// TIA Portal V19 program export: 0 tag tables, 0 data types, 5 data blocks, 88 code blocks (in call order from the OBs), 6 instance data blocks

DATA_BLOCK "DB_System"   // DB3
{ S7_Optimized_Access := 'TRUE' }
// stored: AutoNumber false, MemoryReserve 100
   VAR
      datetime : Struct
         current : DTL := DTL#2025-09-17-14:58:30.265837800;
      END_STRUCT;
      firstCycle : Bool := TRUE;
      reqPointers : Bool := FALSE;
      reqParametrizations : Bool := FALSE;
   END_VAR
   VAR RETAIN
      modulesGroup : Struct
         ADIN { S7_SetPoint := 'True'} : Bool := FALSE;
         AIN { S7_SetPoint := 'True'} : Bool := TRUE;
         DIFF { S7_SetPoint := 'True'} : Bool := FALSE;
         DIN { S7_SetPoint := 'True'} : Bool := TRUE;
         MTR { S7_SetPoint := 'True'} : Bool := TRUE;
         MTRDIR { S7_SetPoint := 'True'} : Bool := TRUE;
         MTRLIN { S7_SetPoint := 'True'} : Bool := FALSE;
         VLV { S7_SetPoint := 'True'} : Bool := FALSE;
         CVLV { S7_SetPoint := 'True'} : Bool := FALSE;
      END_STRUCT;
   END_VAR
   VAR
      reqQuickSetup { S7_SetPoint := 'True'} : "modTypes";
   END_VAR
BEGIN
   reqQuickSetup.adin := FALSE;
   reqQuickSetup.ain := FALSE;
   reqQuickSetup.cvlv := FALSE;
   reqQuickSetup.din := FALSE;
   reqQuickSetup.mtr := FALSE;
   reqQuickSetup.mtrDir := FALSE;
   reqQuickSetup.mtrLin := FALSE;
   reqQuickSetup.vlv := FALSE;
END_DATA_BLOCK

DATA_BLOCK "FAULTS"   // DB14
{ S7_Optimized_Access := 'FALSE' }
   VAR
      ADIN { S7_SetPoint := 'True'} : Array[0.."MAX_ADIN"] of "UDT_DINFAULTS";   // ADIN = 1 alarm/instance, 24 x 8 (each type contains 8 instances) = 192 alarms, offset = 0
      AIN { S7_SetPoint := 'True'} : Array[0.."MAX_AIN"] of "UDT_AINFAULTS";   // AIN = 2 alarms/instance, 200 x 2 = 400 alarms, offset = 192
      DIFF { S7_SetPoint := 'True'} : Array[0.."MAX_DIFF"] of "UDT_AINFAULTS";   // DIFF = 2 alarms/instance, 32 x 2 = 64 alarms, offset = 592
      DIN { S7_SetPoint := 'True'} : Array[0.."MAX_DIN"] of "UDT_DINFAULTS";   // DIN = 1 alarm/instance, 24 x 8 (each type contains 8 instances) = 192 alarms, offset = 656
      MTR { S7_SetPoint := 'True'} : Array[0.."MAX_MTR"] of "UDT_MTRFAULTS";   // MTR = 6 alarms/instance, 200 x 6 = 1200 alarms, offset = 848
      MTRLIN { S7_SetPoint := 'True'} : Array[0.."MAX_MTRLIN"] of "UDT_MTRFAULTS";   // MTRLIN = 6 alarms/instance, 80 x 6 = 480 alarms, offset = 2048
      MTRDIR { S7_SetPoint := 'True'} : Array[0.."MAX_MTRDIR"] of "UDT_MTRFAULTS";   // MTRDIR = 6 alarms/instance, 200 x 6 = 1200 alarms, offset = 2528
      VLV { S7_SetPoint := 'True'} : Array[0.."MAX_VLV"] of "UDT_VALVEFAULTS";   // VLV = 4 alarms/instance, 200 x 6 = 1200 alarms, offset = 3728
      Plant { S7_SetPoint := 'True'} : Array[0.."MAX_PLANT"] of "UDT_DINFAULTS";   // Plant = 1 alarm/instance, 24 x 8 (each type contains 8 instances) = 192 alarms, offset = 4928
   END_VAR
BEGIN
END_DATA_BLOCK

DATA_BLOCK "MODULES_CTRL"   // DB54
{ S7_Optimized_Access := 'TRUE' }
// stored: MemoryReserve 100
   VAR
      ADIN { ExternalAccessible := 'False'; ExternalVisible := 'False'; ExternalWritable := 'False'; S7_SetPoint := 'True'} : Array[0.."M_ADIN"] of "CTRL_ADIN";
      AIN { ExternalAccessible := 'False'; ExternalVisible := 'False'; ExternalWritable := 'False'; S7_SetPoint := 'True'} : Array[0.."M_AIN"] of "CTRL_AIN";
      CVLV { ExternalAccessible := 'False'; ExternalVisible := 'False'; ExternalWritable := 'False'; S7_SetPoint := 'True'} : Array[0.."M_CVLV"] of "CTRL_CVLV";
      DIFF { ExternalAccessible := 'False'; ExternalVisible := 'False'; ExternalWritable := 'False'; S7_SetPoint := 'True'} : Array[0.."M_DIFF"] of "CTRL_DIFF";
      DIN { ExternalAccessible := 'False'; ExternalVisible := 'False'; ExternalWritable := 'False'; S7_SetPoint := 'True'} : Array[0.."M_DIN"] of "CTRL_DIN";
      MTRDIR { ExternalAccessible := 'False'; ExternalVisible := 'False'; ExternalWritable := 'False'; S7_SetPoint := 'True'} : Array[0.."M_MTRDIR"] of "CTRL_MTRDIR";
      MTRLIN { ExternalAccessible := 'False'; ExternalVisible := 'False'; ExternalWritable := 'False'; S7_SetPoint := 'True'} : Array[0.."M_MTRLIN"] of "CTRL_MTRLIN";
      MTR { ExternalAccessible := 'False'; ExternalVisible := 'False'; ExternalWritable := 'False'; S7_SetPoint := 'True'} : Array[0.."M_MTR"] of "CTRL_MTR";
      VLV { ExternalAccessible := 'False'; ExternalVisible := 'False'; ExternalWritable := 'False'; S7_SetPoint := 'True'} : Array[0.."M_VLV"] of "CTRL_VLV";
   END_VAR
BEGIN
END_DATA_BLOCK

DATA_BLOCK "WARNINGS"   // DB15
{ S7_Optimized_Access := 'FALSE' }
   VAR
      AIN { S7_SetPoint := 'True'} : Array[0.."MAX_AIN"] of "UDT_AINWARNS";   // AIN = 2 alarms/instance, 200 x 2 = 400 alarms, offset = 8000
      DIFF { S7_SetPoint := 'True'} : Array[0.."MAX_DIFF"] of "UDT_AINWARNS";   // DIFF = 2 alarms/instance, 200 x 2 = 400 alarms, offset = 8400
      Plant { S7_SetPoint := 'True'} : Array[0.."MAX_PLANT"] of "UDT_DINFAULTS";   // Plant = 1 alarm/instance, 24 x 8 (each type contains 8 instances) = 192 alarms, offset = 8800
   END_VAR
BEGIN
END_DATA_BLOCK

DATA_BLOCK "SpProd"   // DB220
{ S7_Optimized_Access := 'TRUE' }
AUTHOR : CH
FAMILY : Aktina
NAME : SEQUENCE
// stored: AutoNumber false, MemoryReserve 100
   VAR RETAIN
      drill { S7_SetPoint := 'True'} : "dtDrill";
      supply : "dtSupply";
   END_VAR
   VAR
      iTank { S7_SetPoint := 'True'} : Array[0..1] of "UDT_TANKPRESS_2";
      autoReset { S7_SetPoint := 'True'} : Array[0..0] of "dtAutoReset";
   END_VAR
BEGIN
   drill.level[0] := 75;
   drill.level[1] := 85;
   drill.level[2] := 90;
   drill.level[3] := 100;
   drill.tDelay := T#5S;
   drill.setPriority[0] := 2;
   drill.setPriority[1] := 3;
   drill.setPriority[2] := 0;
   drill.loadPriority[0] := 2;
   drill.loadPriority[1] := 3;
   drill.loadPriority[2] := 0;
   drill.TankAvailable[0..1] := TRUE;
   drill.loadBtn := FALSE;
   supply.setAvailPumps[0] := FALSE;
   supply.setAvailPumps[1..3] := TRUE;
   supply.loadAvailPumps[0] := FALSE;
   supply.loadAvailPumps[1..3] := TRUE;
   supply.availPumps[0..2] := TRUE;
   supply.loadBtn := FALSE;
   supply.pressureSP := 4.0;
   supply.hhPressureAlm := 6.0;
   supply.highFlow := 35.0;
   supply.lowFlow := 10.0;
   supply.zChangeThr := 0.3;
   supply.zChangeDelay := T#1S;
   supply.PumpInterval := T#10H;
   supply.zoneChangeOP := 90.0;
   supply.overlapDelay := T#10S;
   supply.downgradeDelay := T#40S;
   supply.chLead := 2;
   supply.enRotation := FALSE;
   supply.stageUp.zoneChangeOP := 95.0;
   supply.stageUp.delayUpgrade := T#5S;
   // supply.stageDown[0] : bigPump
   // supply.stageDown[1] : midPump
   // supply.stageDown[2] : smallPump
   supply.stageDown[0..3].zoneChangeOP := 40.0;
   supply.stageDown[0..3].prevOP := 20.0;
   supply.stageDown[0..3].nextOP := 70.0;
   supply.stageDown[0].stabilizeDelay := T#1M;
   supply.stageDown[1].stabilizeDelay := T#10S;
   supply.stageDown[2..3].stabilizeDelay := T#5S;
   supply.stageDown[0..3].followUp := FALSE;
   iTank[0..1].r := 1.0;
   iTank[0..1].d := 263.0;
   iTank[0..1].hPt := 0.0;
   iTank[0..1].hBase := 0.0;
   iTank[0..1].hCyl := 525.0;
   iTank[0].hAct := 465.6394;
   iTank[1].hAct := 463.0353;
   iTank[0].vol := 25295.94;
   iTank[1].vol := 25154.47;
   // autoReset[0] : Grid
   autoReset[0].maxAlarms := 10;
   autoReset[0].perT := T#1H;
   autoReset[0].autoresetT := T#30S;
END_DATA_BLOCK

ORGANIZATION_BLOCK "Main"   // OB1, LAD, ProgramCycle
TITLE = "Main Program Sweep (Cycle)"
{ S7_Optimized_Access := 'TRUE' }
// stored: SetENOAutomatically false
   VAR_INPUT
      Initial_Call : Bool;   // Initial call of this OB
      Remanence : Bool;   // =True, if remanent data are available
   END_VAR
BEGIN
END_ORGANIZATION_BLOCK

ORGANIZATION_BLOCK "Cyclic interrupt 100ms"   // OB30, LAD, CyclicInterrupt
{ S7_Optimized_Access := 'TRUE' }
// stored: SetENOAutomatically false
   VAR_INPUT
      Initial_Call : Bool;   // Initial call of this OB
      Event_Count : Int;   // Events discarded
   END_VAR
   VAR_TEMP
      i : Int;
   END_VAR
BEGIN
END_ORGANIZATION_BLOCK

ORGANIZATION_BLOCK "Diagnostic error interrupt"   // OB82, LAD, DiagnosticErrorInterrupt
{ S7_Optimized_Access := 'TRUE' }
// stored: SetENOAutomatically false
   VAR_INPUT
      IO_State : Word;   // IO state of the HW object
      LADDR : HW_ANY;   // Hardware identifier
      Channel : UInt;   // Channel number
      MultiError : Bool;   // =true if more than one error is present
   END_VAR
BEGIN
END_ORGANIZATION_BLOCK

ORGANIZATION_BLOCK "Pull or plug of modules"   // OB83, LAD, PullOrPlugOfModules
{ S7_Optimized_Access := 'TRUE' }
// stored: SetENOAutomatically false
   VAR_INPUT
      LADDR : HW_IO;   // Hardware identifier
      Event_Class : Byte;   // 16#38/39: module inserted, removed
      Fault_ID : Byte;   // Fault identifier
   END_VAR
BEGIN
END_ORGANIZATION_BLOCK

ORGANIZATION_BLOCK "Rack or station failure"   // OB86, LAD, RackOrStationFailure
{ S7_Optimized_Access := 'TRUE' }
// stored: SetENOAutomatically false
   VAR_INPUT
      LADDR : HW_DEVICE;   // Hardware identifier
      Event_Class : Byte;   // Event class
      Fault_ID : Byte;   // Fault identifier
   END_VAR
BEGIN
END_ORGANIZATION_BLOCK

ORGANIZATION_BLOCK "Time error interrupt"   // OB80, LAD, TimeErrorInterrupt
{ S7_Optimized_Access := 'TRUE' }
// stored: SetENOAutomatically false
   VAR_INPUT
      Fault_ID : Byte;   // Fault identifier
      Csg_OBnr : OB_ANY;   // Number of OB causing the error
      Csg_Prio : UInt;   // Priority of OB causing the error
   END_VAR
BEGIN
END_ORGANIZATION_BLOCK

FUNCTION_BLOCK "AFB_Totalizer"   // FB3, LAD
{ S7_Optimized_Access := 'TRUE' }
// stored: MemoryReserve 100, SetENOAutomatically false
   VAR_INPUT
      inputVolume { ExternalAccessible := 'False'; ExternalVisible := 'False'; ExternalWritable := 'False'} : Real;
      startBtn { ExternalAccessible := 'False'; ExternalVisible := 'False'; ExternalWritable := 'False'} : Bool;
      stopBtn { ExternalAccessible := 'False'; ExternalVisible := 'False'; ExternalWritable := 'False'} : Bool;
   END_VAR
   VAR_OUTPUT
      addedVolume { ExternalAccessible := 'False'; ExternalVisible := 'False'; ExternalWritable := 'False'} : Real;
      tempCount { ExternalAccessible := 'False'; ExternalVisible := 'False'; ExternalWritable := 'False'} : Bool;
   END_VAR
   VAR
      previousVolume { ExternalAccessible := 'False'; ExternalVisible := 'False'; ExternalWritable := 'False'} : Real;
      Start_Trigger { S7_SetPoint := 'True'} : R_TRIG;
      Strop_Trigger { S7_SetPoint := 'True'} : R_TRIG;
   END_VAR
BEGIN

REGION Network 1
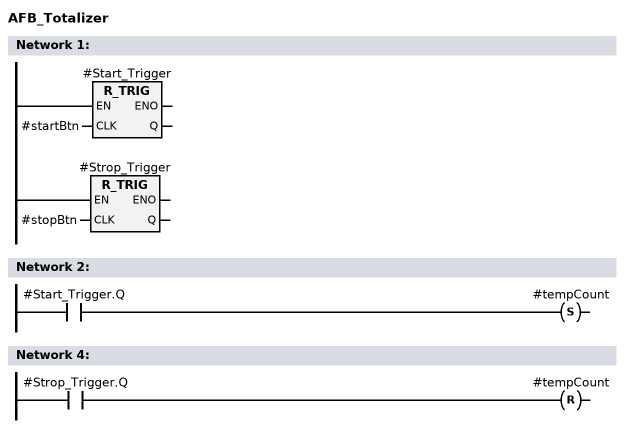
   RUNG wire#powerrail
      #Start_Trigger.R_TRIG(CLK := #startBtn, Q =>)
   END_RUNG
   RUNG wire#powerrail
      #Strop_Trigger.R_TRIG(CLK := #stopBtn, Q =>)
   END_RUNG
   // the same network as SCL:
   #Start_Trigger(CLK := #startBtn);   // R_TRIG
   #Strop_Trigger(CLK := #stopBtn);   // R_TRIG
END_REGION

REGION Network 2
   RUNG wire#powerrail
      Contact( #Start_Trigger.Q )
      S_Coil( #tempCount )
   END_RUNG
   // the same network as SCL:
   IF #Start_Trigger.Q THEN #tempCount := TRUE; END_IF;
END_REGION

REGION Network 3 (SCL)

   IF #startBtn THEN
       #previousVolume := #inputVolume;
   END_IF;


   IF #tempCount THEN

       #addedVolume := #inputVolume - #previousVolume;
       ;
   ELSE
       #addedVolume := 0 ;
   END_IF;
END_REGION

REGION Network 4
   RUNG wire#powerrail
      Contact( #Strop_Trigger.Q )
      R_Coil( #tempCount )
   END_RUNG
   // the same network as SCL:
   IF #Strop_Trigger.Q THEN #tempCount := FALSE; END_IF;
END_REGION
END_FUNCTION_BLOCK

FUNCTION "AFC_Counter" : Void   // FC1, FBD
TITLE = AFC_COUNTER
{ S7_Optimized_Access := 'TRUE' }
AUTHOR : CH
FAMILY : Aktina
NAME : Global
// AFC_COUNTER
// stored: AutoNumber false, IsIECCheckEnabled true, SetENOAutomatically false
   VAR_INPUT
      Trigger : Bool;
      Pulse : Bool;
      Reset : Bool;
   END_VAR
   VAR_IN_OUT
      Data : Variant;
   END_VAR
   VAR_TEMP
      i : "UDT_COUNTER";
      logical1 : Bool;
   END_VAR
BEGIN

REGION Network 1: GEN: Set Logical 1
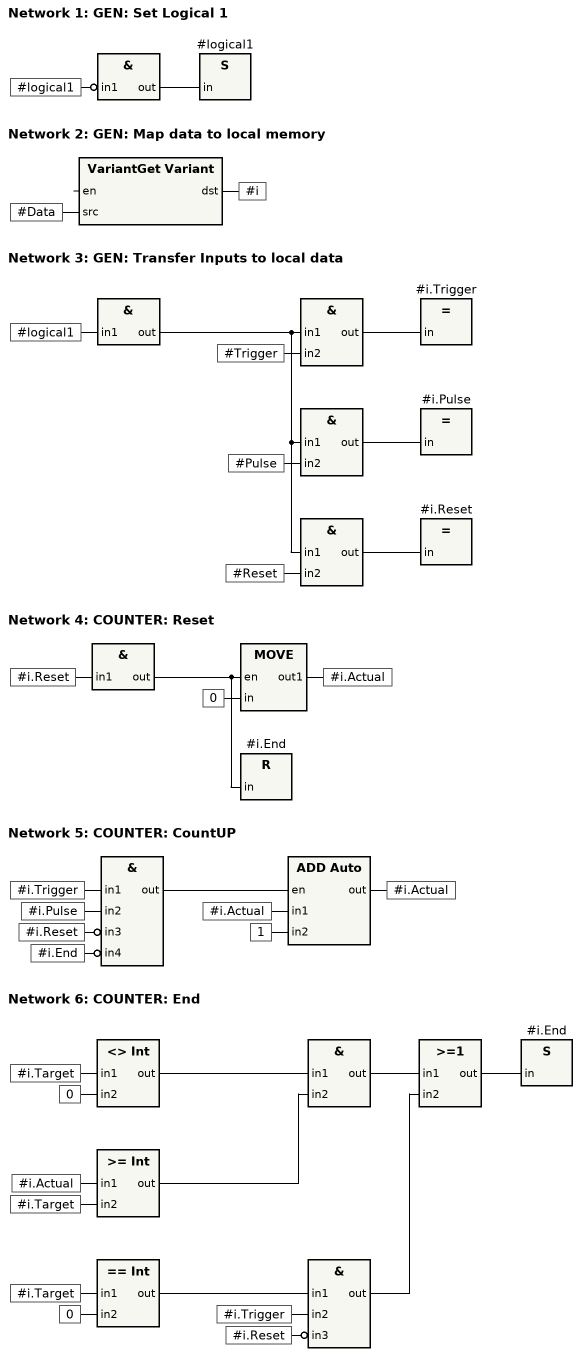
   IF NOT #logical1 THEN #logical1 := TRUE; END_IF;
END_REGION

REGION Network 2: GEN: Map data to local memory
   // no SCL statement known for VariantGet: written as a call
   VariantGet(src := #Data, dst => #i);
END_REGION

REGION Network 3: GEN: Transfer Inputs to local data
   #i.Trigger := #logical1 AND #Trigger;
   #i.Pulse := #logical1 AND #Pulse;
   #i.Reset := #logical1 AND #Reset;
END_REGION

REGION Network 4: COUNTER: Reset
   IF #i.Reset THEN
       #i.Actual := 0;
       #i.End := FALSE;
   END_IF;
END_REGION

REGION Network 5: COUNTER: CountUP
   IF #i.Trigger AND #i.Pulse AND NOT #i.Reset AND NOT #i.End THEN #i.Actual := #i.Actual + 1; END_IF;
END_REGION

REGION Network 6: COUNTER: End
   IF ((#i.Target <> 0) AND (#i.Actual >= #i.Target)) OR ((#i.Target = 0) AND #i.Trigger AND NOT #i.Reset) THEN
       #i.End := TRUE;
   END_IF;
END_REGION

REGION Network 7: COUNTER: Calculate Remaining
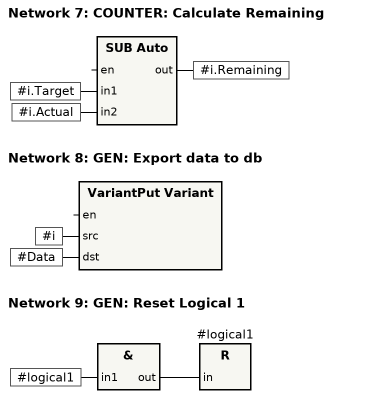
   #i.Remaining := #i.Target - #i.Actual;
END_REGION

REGION Network 8: GEN: Export data to db
   // no SCL statement known for VariantPut: written as a call
   VariantPut(src := #i, dst := #Data);
END_REGION

REGION Network 9: GEN: Reset Logical 1
   IF #logical1 THEN #logical1 := FALSE; END_IF;
END_REGION
END_FUNCTION

FUNCTION "AFC_DelayON" : Void   // FC2, FBD
TITLE = AFC_DELAYON
{ S7_Optimized_Access := 'TRUE' }
AUTHOR : CH
FAMILY : Aktina
NAME : Global
// AFC_DELAYON
// stored: AutoNumber false, IsIECCheckEnabled true, SetENOAutomatically false
   VAR_INPUT
      cmd : Bool;   // Command run
      Pulse : Bool;   // 100ms pulse
      Reset : Bool;   // Reset immediately
   END_VAR
   VAR_OUTPUT
      on : Bool;   // Activation
   END_VAR
   VAR_IN_OUT
      Data : Variant;   // Data area
   END_VAR
   VAR_TEMP
      i : "UDT_DELAYON";   // Local stack
      logical1 : Bool;   // Logical 1
      calc : Real;   // Calculation intermediate
   END_VAR
BEGIN

REGION Network 1: GEN: Set Logical 1
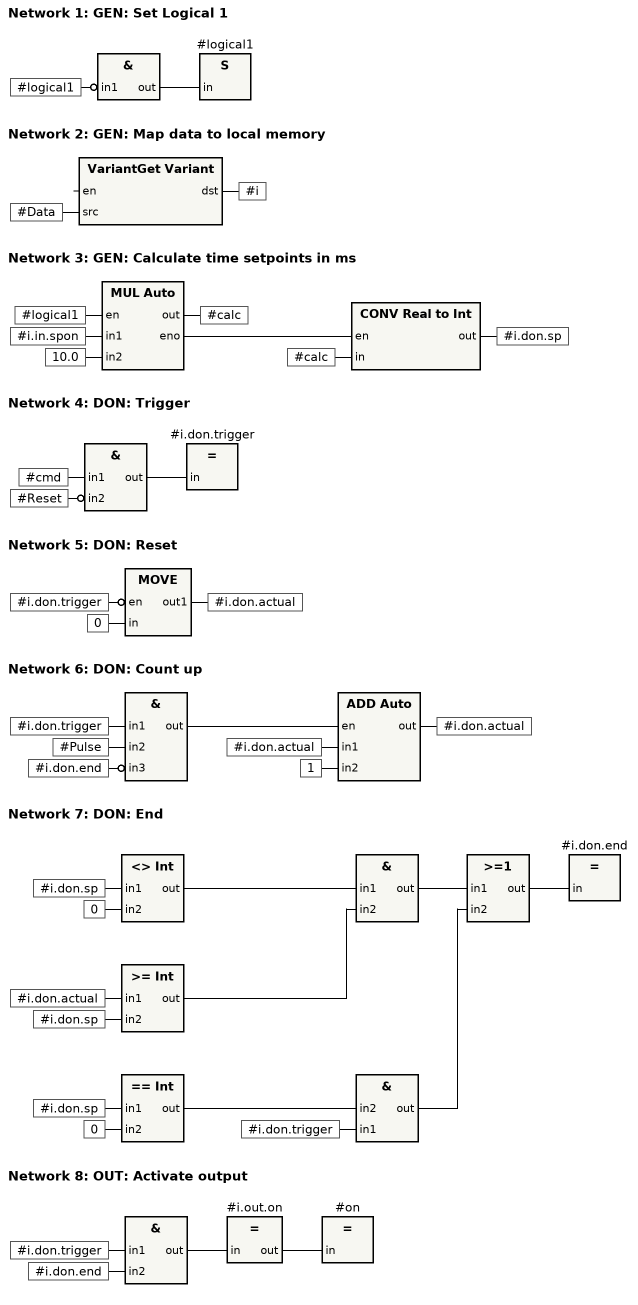
   IF NOT #logical1 THEN #logical1 := TRUE; END_IF;
END_REGION

REGION Network 2: GEN: Map data to local memory
   // no SCL statement known for VariantGet: written as a call
   VariantGet(src := #Data, dst => #i);
END_REGION

REGION Network 3: GEN: Calculate time setpoints in ms
   IF #logical1 THEN
       #calc := #i.in.spon * 10.0;
       #i.don.sp := REAL_TO_INT(#calc);
   END_IF;
END_REGION

REGION Network 4: DON: Trigger
   #i.don.trigger := #cmd AND NOT #Reset;
END_REGION

REGION Network 5: DON: Reset
   IF NOT #i.don.trigger THEN #i.don.actual := 0; END_IF;
END_REGION

REGION Network 6: DON: Count up
   IF #i.don.trigger AND #Pulse AND NOT #i.don.end THEN #i.don.actual := #i.don.actual + 1; END_IF;
END_REGION

REGION Network 7: DON: End
   #i.don.end := ((#i.don.sp <> 0) AND (#i.don.actual >= #i.don.sp)) OR ((#i.don.sp = 0) AND #i.don.trigger);
END_REGION

REGION Network 8: OUT: Activate output
   #i.out.on := #i.don.trigger AND #i.don.end;
   #on := #i.out.on;
END_REGION

REGION Network 9: GEN: Export data to db
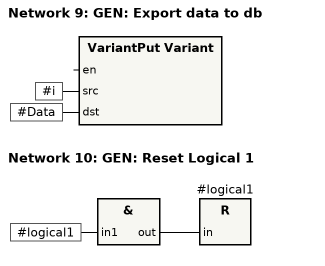
   // no SCL statement known for VariantPut: written as a call
   VariantPut(src := #i, dst := #Data);
END_REGION

REGION Network 10: GEN: Reset Logical 1
   IF #logical1 THEN #logical1 := FALSE; END_IF;
END_REGION
END_FUNCTION

FUNCTION "AFC_DelayONOFF" : Void   // FC4, FBD
TITLE = AFC_DELAYONOFF
{ S7_Optimized_Access := 'TRUE' }
AUTHOR : CH
FAMILY : Aktina
NAME : Global
// AFC_DELAYONOFF
// stored: AutoNumber false, IsIECCheckEnabled true, SetENOAutomatically false
   VAR_INPUT
      cmd : Bool;   // Command run
      Pulse : Bool;   // 100ms pulse
      Reset : Bool;   // Reset immediately
   END_VAR
   VAR_OUTPUT
      on : Bool;   // Activation
   END_VAR
   VAR_IN_OUT
      Data : Variant;   // Data area
   END_VAR
   VAR_TEMP
      i : "UDT_DELAYONOFF";   // Local stack
      logical1 : Bool;   // Logical 1
      calc : Real;   // Calculation intermediate
   END_VAR
BEGIN

REGION Network 1: GEN: Set Logical 1
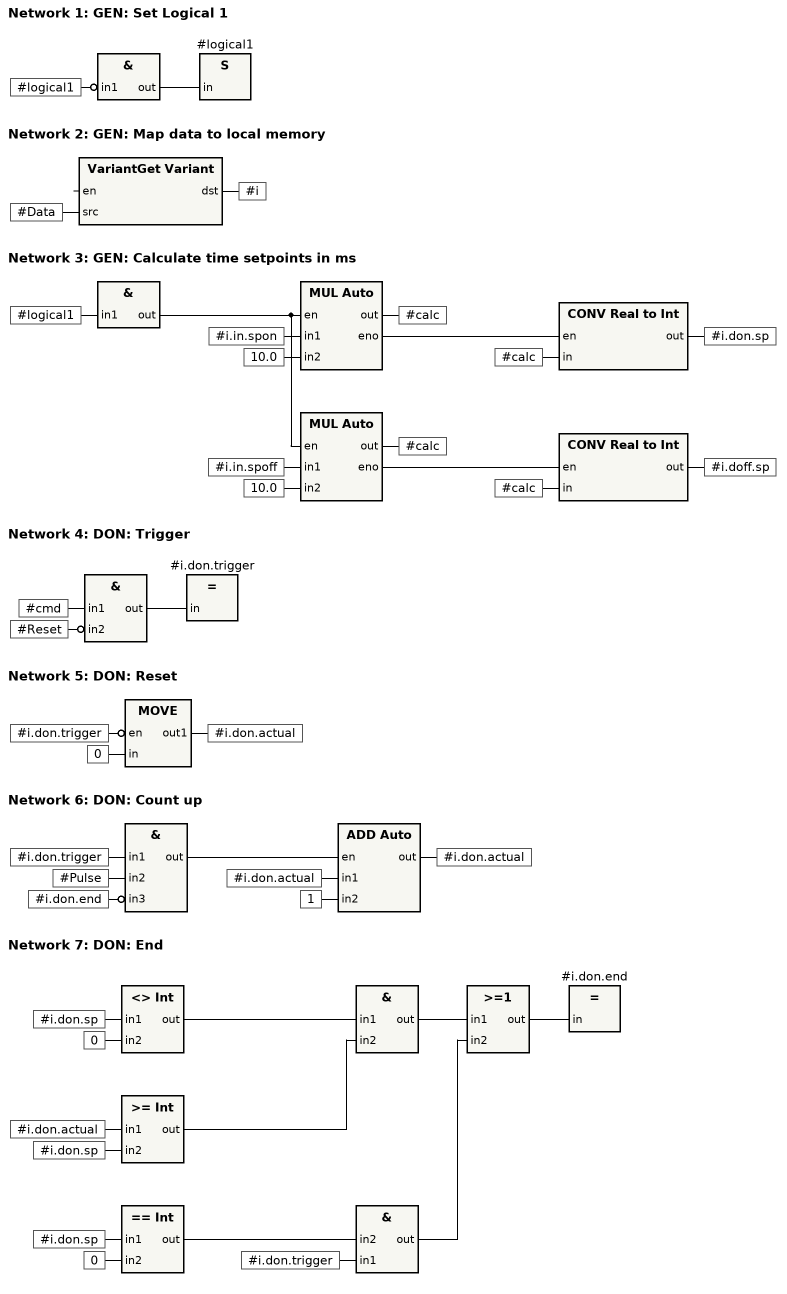
   IF NOT #logical1 THEN #logical1 := TRUE; END_IF;
END_REGION

REGION Network 2: GEN: Map data to local memory
   // no SCL statement known for VariantGet: written as a call
   VariantGet(src := #Data, dst => #i);
END_REGION

REGION Network 3: GEN: Calculate time setpoints in ms
   IF #logical1 THEN
       #calc := #i.in.spon * 10.0;
       #i.don.sp := REAL_TO_INT(#calc);
       #calc := #i.in.spoff * 10.0;
       #i.doff.sp := REAL_TO_INT(#calc);
   END_IF;
END_REGION

REGION Network 4: DON: Trigger
   #i.don.trigger := #cmd AND NOT #Reset;
END_REGION

REGION Network 5: DON: Reset
   IF NOT #i.don.trigger THEN #i.don.actual := 0; END_IF;
END_REGION

REGION Network 6: DON: Count up
   IF #i.don.trigger AND #Pulse AND NOT #i.don.end THEN #i.don.actual := #i.don.actual + 1; END_IF;
END_REGION

REGION Network 7: DON: End
   #i.don.end := ((#i.don.sp <> 0) AND (#i.don.actual >= #i.don.sp)) OR ((#i.don.sp = 0) AND #i.don.trigger);
END_REGION

REGION Network 8: DOFF: Trigger
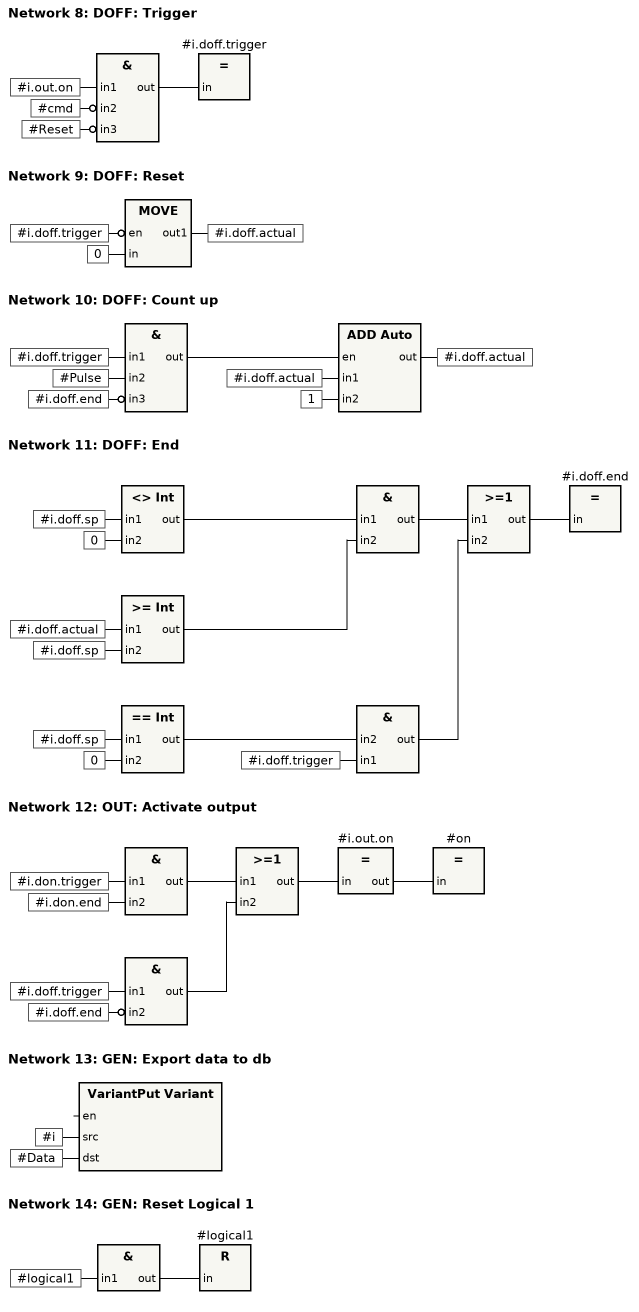
   #i.doff.trigger := #i.out.on AND NOT #cmd AND NOT #Reset;
END_REGION

REGION Network 9: DOFF: Reset
   IF NOT #i.doff.trigger THEN #i.doff.actual := 0; END_IF;
END_REGION

REGION Network 10: DOFF: Count up
   IF #i.doff.trigger AND #Pulse AND NOT #i.doff.end THEN #i.doff.actual := #i.doff.actual + 1; END_IF;
END_REGION

REGION Network 11: DOFF: End
   #i.doff.end := ((#i.doff.sp <> 0) AND (#i.doff.actual >= #i.doff.sp)) OR ((#i.doff.sp = 0) AND #i.doff.trigger);
END_REGION

REGION Network 12: OUT: Activate output
   #i.out.on := (#i.don.trigger AND #i.don.end) OR (#i.doff.trigger AND NOT #i.doff.end);
   #on := #i.out.on;
END_REGION

REGION Network 13: GEN: Export data to db
   // no SCL statement known for VariantPut: written as a call
   VariantPut(src := #i, dst := #Data);
END_REGION

REGION Network 14: GEN: Reset Logical 1
   IF #logical1 THEN #logical1 := FALSE; END_IF;
END_REGION
END_FUNCTION

FUNCTION "AFC_Steptimer" : Void   // FC35, FBD
TITLE = AFC_Steptimer
{ S7_Optimized_Access := 'TRUE' }
AUTHOR : CH
FAMILY : Aktina
NAME : Global
// AFC_Steptimer
// stored: AutoNumber false, SetENOAutomatically false
   VAR_INPUT
      "step" : Bool;   // Step activated
      count_max : Bool;   // Trigger for max step timer
      count_step : Bool;   // Trigger for conditional step timer
      Pulse : Bool;   // Pulse used for time count
      reset_max : Bool;   // Reset max step timer
      reset_step : Bool;   // Reset conditional step timer
      reset_warn : Bool;   // Reset max timer warning
   END_VAR
   VAR_OUTPUT
      max_warn : Bool;   // Max step timer has elapsed
   END_VAR
   VAR_IN_OUT
      Data : Variant;   // Unique data area for this counter
   END_VAR
   VAR_TEMP
      i : "UDT_STEPTIMER";
      logical1 : Bool;
      remain : UDInt;
      intermediate : UDInt;
      sec : UDInt;
      min : UDInt;
      hour : UDInt;
   END_VAR
BEGIN

REGION Network 1: GEN: Create Logical 1
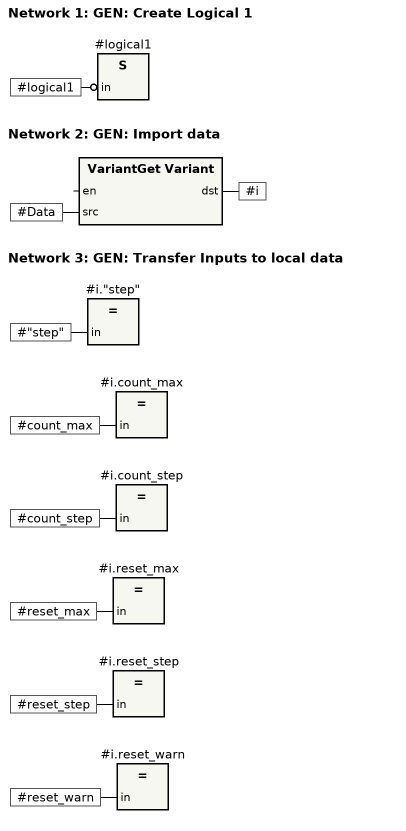
   IF NOT #logical1 THEN #logical1 := TRUE; END_IF;
END_REGION

REGION Network 2: GEN: Import data
   // no SCL statement known for VariantGet: written as a call
   VariantGet(src := #Data, dst => #i);
END_REGION

REGION Network 3: GEN: Transfer Inputs to local data
   #i."step" := #"step";
   #i.count_max := #count_max;
   #i.count_step := #count_step;
   #i.reset_max := #reset_max;
   #i.reset_step := #reset_step;
   #i.reset_warn := #reset_warn;
END_REGION

REGION Network 4: TIMER: Calculate seconds based on h, m, s (max)
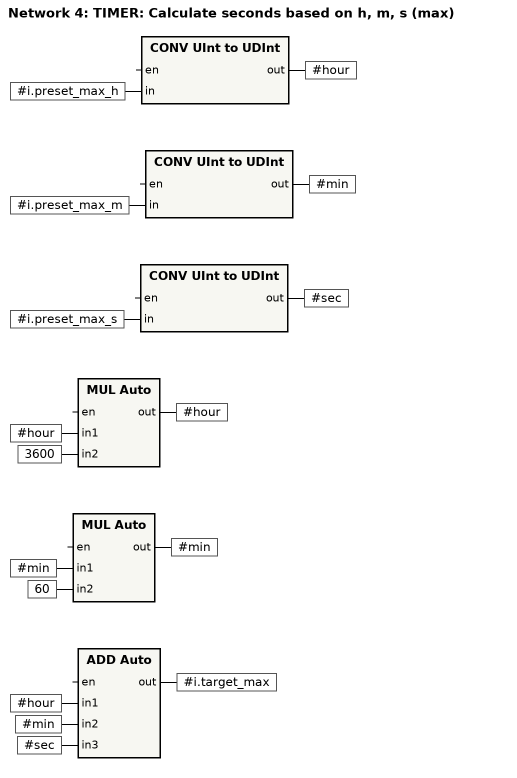
   #hour := UINT_TO_UDINT(#i.preset_max_h);
   #min := UINT_TO_UDINT(#i.preset_max_m);
   #sec := UINT_TO_UDINT(#i.preset_max_s);
   #hour := #hour * 3600;
   #min := #min * 60;
   #i.target_max := #hour + #min + #sec;
END_REGION

REGION Network 5: TIMER: Calculate seconds based on h, m, s (step)
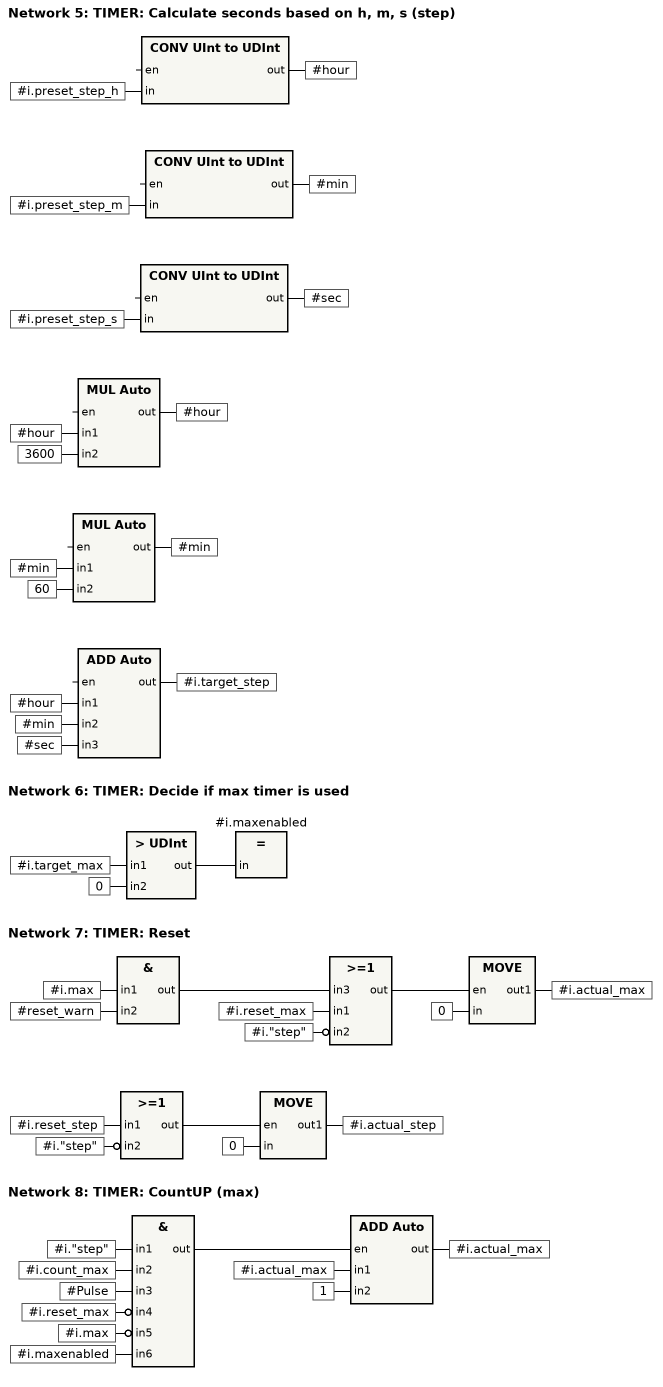
   #hour := UINT_TO_UDINT(#i.preset_step_h);
   #min := UINT_TO_UDINT(#i.preset_step_m);
   #sec := UINT_TO_UDINT(#i.preset_step_s);
   #hour := #hour * 3600;
   #min := #min * 60;
   #i.target_step := #hour + #min + #sec;
END_REGION

REGION Network 6: TIMER: Decide if max timer is used
   #i.maxenabled := #i.target_max > 0;
END_REGION

REGION Network 7: TIMER: Reset
   IF (#i.max AND #reset_warn) OR #i.reset_max OR NOT #i."step" THEN #i.actual_max := 0; END_IF;
   IF #i.reset_step OR NOT #i."step" THEN #i.actual_step := 0; END_IF;
END_REGION

REGION Network 8: TIMER: CountUP (max)
   IF #i."step" AND #i.count_max AND #Pulse AND NOT #i.reset_max AND NOT #i.max AND #i.maxenabled THEN
       #i.actual_max := #i.actual_max + 1;
   END_IF;
END_REGION

REGION Network 9: TIMER: CountUP (step)
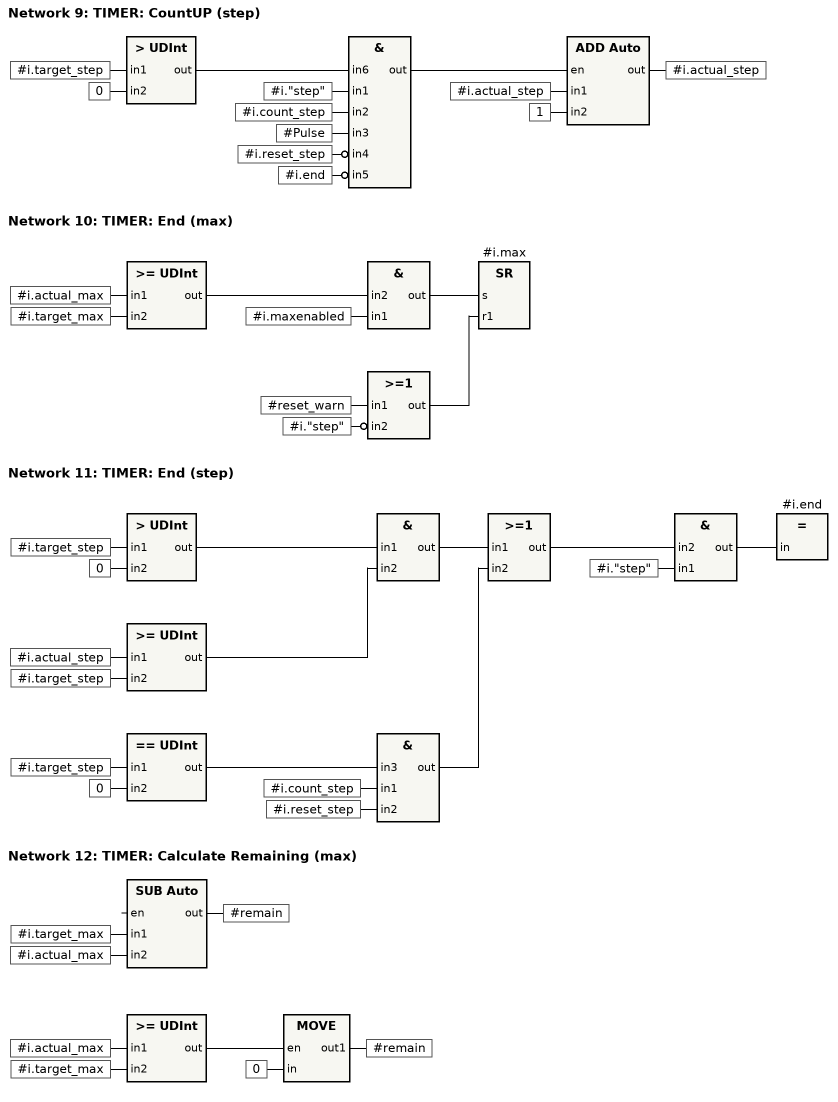
   IF (#i.target_step > 0) AND #i."step" AND #i.count_step AND #Pulse AND NOT #i.reset_step AND NOT #i.end THEN
       #i.actual_step := #i.actual_step + 1;
   END_IF;
END_REGION

REGION Network 10: TIMER: End (max)
   IF (#i.actual_max >= #i.target_max) AND #i.maxenabled THEN
       #i.max := TRUE;   // SR flip-flop
   END_IF;
   IF #reset_warn OR NOT #i."step" THEN #i.max := FALSE; END_IF;
END_REGION

REGION Network 11: TIMER: End (step)
   #i.end := (((#i.target_step > 0) AND (#i.actual_step >= #i.target_step)) OR ((#i.target_step = 0) AND #i.count_step AND #i.reset_step)) AND #i."step";
END_REGION

REGION Network 12: TIMER: Calculate Remaining (max)
   #remain := #i.target_max - #i.actual_max;
   IF #i.actual_max >= #i.target_max THEN #remain := 0; END_IF;
END_REGION

REGION Network 13: TIMER: Convert remaining to h, m, s (max)
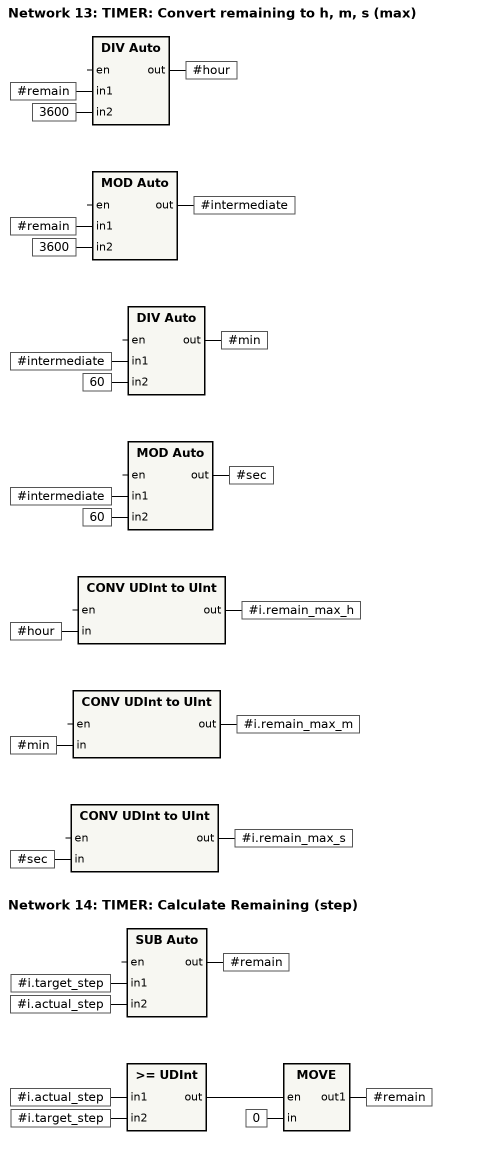
   #hour := #remain / 3600;
   #intermediate := #remain MOD 3600;
   #min := #intermediate / 60;
   #sec := #intermediate MOD 60;
   #i.remain_max_h := UDINT_TO_UINT(#hour);
   #i.remain_max_m := UDINT_TO_UINT(#min);
   #i.remain_max_s := UDINT_TO_UINT(#sec);
END_REGION

REGION Network 14: TIMER: Calculate Remaining (step)
   #remain := #i.target_step - #i.actual_step;
   IF #i.actual_step >= #i.target_step THEN #remain := 0; END_IF;
END_REGION

REGION Network 15: TIMER: Convert remaining to h, m, s (step)
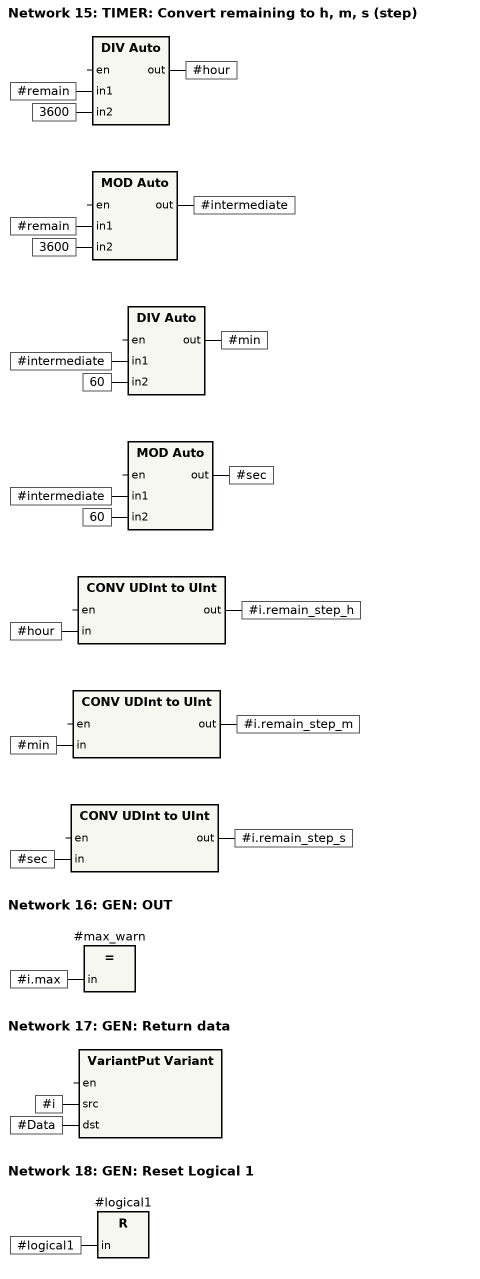
   #hour := #remain / 3600;
   #intermediate := #remain MOD 3600;
   #min := #intermediate / 60;
   #sec := #intermediate MOD 60;
   #i.remain_step_h := UDINT_TO_UINT(#hour);
   #i.remain_step_m := UDINT_TO_UINT(#min);
   #i.remain_step_s := UDINT_TO_UINT(#sec);
END_REGION

REGION Network 16: GEN: OUT
   #max_warn := #i.max;
END_REGION

REGION Network 17: GEN: Return data
   // no SCL statement known for VariantPut: written as a call
   VariantPut(src := #i, dst := #Data);
END_REGION

REGION Network 18: GEN: Reset Logical 1
   IF #logical1 THEN #logical1 := FALSE; END_IF;
END_REGION
END_FUNCTION

FUNCTION "Manager" : Void   // FC201, LAD
{ S7_Optimized_Access := 'TRUE' }
AUTHOR : CH
FAMILY : Aktina
NAME : PROCESS
// stored: AutoNumber false, SetENOAutomatically false
   VAR CONSTANT
      maxVol : Real := 45359.24;
   END_VAR
BEGIN

REGION Network 1 (SCL): Tank mbar to vol
END_REGION

REGION Network 2 (SCL): // Process Function
END_REGION
END_FUNCTION

ORGANIZATION_BLOCK "Startup"
TITLE = "Complete Restart"
{ S7_Optimized_Access := 'TRUE' }
VERSION : 0.1

BEGIN
	"DB_System".firstCycle := TRUE;
END_ORGANIZATION_BLOCK

FUNCTION_BLOCK "AFB_ADIN_v3"
{ S7_Optimized_Access := 'TRUE' }
VERSION : 0.1
   VAR_INPUT 
      input { ExternalAccessible := 'False'; ExternalVisible := 'False'; ExternalWritable := 'False'} : Real;   // Analog sensor value to be compared
      monitorfault { ExternalAccessible := 'False'; ExternalVisible := 'False'; ExternalWritable := 'False'} : Bool;   // Release fault monitoring
      p1s { ExternalAccessible := 'False'; ExternalVisible := 'False'; ExternalWritable := 'False'} : Bool;   // Pulse edge for 1Hz
      p100ms { ExternalAccessible := 'False'; ExternalVisible := 'False'; ExternalWritable := 'False'} : Bool;   // Pulse edge for 10Hz
      generalackn { ExternalAccessible := 'False'; ExternalVisible := 'False'; ExternalWritable := 'False'} : Bool;   // General acknowledgement
      reset { ExternalAccessible := 'False'; ExternalVisible := 'False'; ExternalWritable := 'False'} : Bool;   // Reset Fault
      mute { ExternalAccessible := 'False'; ExternalVisible := 'False'; ExternalWritable := 'False'} : Bool;   // Mute siren
      Unit { ExternalAccessible := 'False'; ExternalVisible := 'False'; ExternalWritable := 'False'} : WString;   // Analog sensor's unit
   END_VAR

   VAR_OUTPUT 
      Switch { ExternalAccessible := 'False'; ExternalVisible := 'False'; ExternalWritable := 'False'} : Bool;   // Switch after time cross check
   END_VAR

   VAR_IN_OUT 
      alarm_adin { ExternalAccessible := 'False'; ExternalVisible := 'False'; ExternalWritable := 'False'} : Bool;
      plcackn_adin { ExternalAccessible := 'False'; ExternalVisible := 'False'; ExternalWritable := 'False'} : Bool;
      siren_adin { ExternalAccessible := 'False'; ExternalVisible := 'False'; ExternalWritable := 'False'} : Bool;
      hmiackn_adin { ExternalAccessible := 'False'; ExternalVisible := 'False'; ExternalWritable := 'False'} : Bool;
   END_VAR

   VAR RETAIN
      i : "UDT_ADIN";   // UDT containing scale process data
   END_VAR

   VAR_TEMP 
      condSET : Bool;
      condRESET : Bool;
   END_VAR


BEGIN
	REGION SIM NW:2-3
	    
	    // Network2: SIM: Simulation
	
	    #i.sim.simulated := (#i.sim.simulated OR #i.sim.cmdon) AND NOT #i.sim.cmdoff;
	    
	    // Network3: SIM: Force
	    
	    #condSET := #i.sim.cmdforce;
	    #condRESET := #i.sim.cmdunforce OR (NOT #i.sim.simulated);
	    
	    #i.sim.forced := (#i.sim.forced OR #condSET) AND NOT #condRESET;
	    
	END_REGION
	
	REGION STATUS: NW:4-6
	    
	    // Network4: STATUS: Raw input
	    
	    #i.status.rawinput := #input;
	    
	    // Network5: STATUS: Processed input
	    
	    #i.status.processed := ((#i.status.rawinput > #i.setup.reference) AND (#i.setup.comparison = 0)) OR
	                            ((#i.status.rawinput >= #i.setup.reference) AND (#i.setup.comparison = 1)) OR
	                            ((#i.status.rawinput < #i.setup.reference) AND (#i.setup.comparison = 2)) OR
	                            ((#i.status.rawinput <= #i.setup.reference) AND (#i.setup.comparison = 3));
	
	    // Network6: STATUS: Alarm monitor     
	    
	    #i.status.alarm_monitor := #monitorfault AND #i.faults.adin.setup."en";
	    
	END_REGION
	
	REGION ADIN: NW 7-9
	    
	    // Network7: ADIN: Reset actual timers
	    
	    IF #i.sim.simulated OR (#i.status.processed AND #i.status.switch_active) THEN
	        
	        #i."time".on_act := #i."time".off_act := 0;
	        
	    END_IF;
	    
	    IF #i.sim.simulated OR (NOT #i.status.processed AND NOT #i.status.switch_active) THEN
	        
	        #i."time".on_act := #i."time".off_act := 0;
	        
	    END_IF;
	    
	    
	    // Network8: ADIN: Counter
	    
	    IF (#i.status.processed AND NOT #i.status.switch_active) AND #p1s THEN
	        
	        #i."time".on_act := #i."time".on_act + 1;
	        
	    END_IF;
	    
	    IF (NOT #i.status.processed AND #i.status.switch_active) AND #p1s THEN
	        
	        #i."time".off_act := #i."time".off_act + 1;
	        
	    END_IF;
	    
	    // Network9: ADIN: Set switch active
	    
	    #condSET := #i.sim.forced OR (#i.status.processed AND NOT #i.sim.simulated AND (#i."time".on_act >= #i."time".on_set));
	    #condRESET := (NOT #i.sim.forced AND #i.sim.simulated) OR (NOT #i.status.processed AND NOT #i.sim.simulated AND (#i."time".off_act >= #i."time".off_set));
	    
	    #i.status.switch_active := (#i.status.switch_active OR #condSET) AND NOT #condRESET;
	    
	END_REGION
	
	REGION FAULT: NW 10
	    
	    // Network10: FAULT: Switch activated
	    
	    "AFC_AlarmAckn"(trigger:=(NOT #i.setup.triggerversion AND NOT #i.status.switch_active) OR ((#i.setup.triggerversion AND #i.status.switch_active)),
	                    release:=#monitorfault,
	                    ctrlpoint:=FALSE,
	                    enackn:=TRUE,
	                    ensiren:=TRUE,
	                    p100ms:=#p100ms,
	                    generalackn:=#generalackn OR #i.faults.fpreset,
	                    reset:=#reset OR #i.faults.fpreset,
	                    mute:=#mute,
	                    delay:=0.0,
	                    plcackn=>#plcackn_adin,
	                    alarm=>#alarm_adin,
	                    siren=>#siren_adin,
	                    hmiackn:=#hmiackn_adin,
	                    Data:=#i.faults.adin);
	    
	END_REGION
	
	REGION GEN: NW 11-12
	    
	    // Network11: FAULT: Switch activated
	    
	    #Switch := #i.status.switch_active;
	    
	    // Network12: FAULT: Switch activated - @CH: This network is provided to treat the phenomenon of non-reset buttons
	    
	    IF #i.faults.fpreset THEN
	        
	        #i.faults.fpreset := FALSE;
	        
	    END_IF;
	    
	END_REGION
END_FUNCTION_BLOCK

FUNCTION "AFC_AlarmAckn" : Void
TITLE = AFC_ALARMACKN
{ S7_Optimized_Access := 'TRUE' }
AUTHOR : CH
FAMILY : Aktina
NAME : Global
VERSION : 0.1
//AFC_ALARMACKN
   VAR_INPUT 
      trigger : Bool;   // Alarm trigger
      release : Bool;   // Release alarm
      ctrlpoint : Bool;   // Control point (0=HMI, 1=PLC)
      enackn : Bool;   // Enable acknowledgement (0=disable, 1=enable)
      ensiren : Bool;   // Enable siren for this alarm
      p100ms : Bool;   // 100ms pulse
      generalackn : Bool;   // General acknowledgement
      reset : Bool;   // Reset
      mute : Bool;   // Mute siren
      delay : Real;   // Delay on (s)
   END_VAR

   VAR_OUTPUT 
      plcackn : Bool;   // PLC acknowledgement bit
      alarm : Bool;   // Activation
      siren : Bool;   // Siren
   END_VAR

   VAR_IN_OUT 
      hmiackn : Bool;   // HMI acknowledgement bit
      Data : Variant;   // UDT symbolic address in global DB
   END_VAR

   VAR_TEMP 
      i : "UDT_ALARMACKN";   // Data processed in local memory
   END_VAR


BEGIN
	
	(*Import data*)
	VariantGet(SRC:=#Data,
	           DST=>#i);
	
	(*Calculate setpoint*)
	IF #ctrlpoint THEN
	    #i.setup."en" := #release;
	    #i.don.sp := REAL_TO_UINT(#delay * 10.0);
	ELSE
	    #i.don.sp := REAL_TO_UINT(#i.setup.spon * 10.0);
	END_IF;
	
	// (*PLC acknowledgement*)
	// IF #enackn AND #i.status.alarm THEN
	//     IF #hmiackn OR #generalackn THEN
	//         #i.status.plcackn := TRUE;
	//     END_IF;
	// ELSE
	//     #hmiackn := #i.status.plcackn := FALSE;
	// END_IF;
	
	
	(*PLC acknowledgement*)
	IF #enackn AND #i.status.alarm THEN
	    IF (*#hmiackn OR*)#generalackn THEN
	        #i.status.plcackn := TRUE;
	    END_IF;
	ELSE
	    (*#hmiackn :=*) 
	    #i.status.plcackn := FALSE;
	END_IF;
	
	(*Reset counter*)
	IF NOT #trigger OR #i.status.alarm OR NOT #release OR NOT #i.setup."en" OR (#i.setup.spon = 0.0)  THEN
	    #i.don.actual := 0;
	END_IF;
	
	(*Alarming function*)
	IF #release AND #i.setup."en" AND (#i.setup.spon > 0.0)  THEN
	    
	    (*Count-up*)
	    #i.don.countup := #trigger AND #i.don.actual < #i.don.sp;
	    
	    IF #i.don.countup AND #p100ms AND NOT #i.don.end THEN
	        #i.don.actual := #i.don.actual + 1;
	    END_IF;
	    
	    (*Alarm & Siren generation*)
	    IF #trigger AND #i.don.actual >= #i.don.sp THEN
	        
	        IF #ensiren AND NOT #i.status.alarm THEN
	            #i.status.siren := TRUE;
	        END_IF;
	        #i.status.alarm := TRUE;
	    END_IF;
	    
	    (*Siren reset*)
	    IF NOT #ensiren OR #mute OR #i.status.plcackn OR NOT #i.status.alarm THEN
	        #i.status.siren := FALSE;
	    END_IF;
	    
	    (*Alarm reset*)
	    IF NOT #trigger AND #i.status.alarm AND ((#enackn AND #i.status.plcackn) OR NOT #enackn) AND #reset THEN
	        #i.status.alarm := FALSE;
	    END_IF;
	    
	    
	ELSE
	    #i.status.alarm :=  #i.status.siren := #i.don.countup := (*#hmiackn :=*) #i.status.plcackn := FALSE;
	END_IF;
	    
	#plcackn := #i.status.plcackn;
	#alarm := #i.status.alarm;
	#siren := #i.status.siren;
	
	    (*Export data*)
	    VariantPut(SRC:=#i,
	               DST:=#Data);
	    
	    RETURN;
END_FUNCTION

FUNCTION_BLOCK "AFB_AIN_v3"
{ S7_Optimized_Access := 'TRUE' }
VERSION : 0.1
   VAR_INPUT 
      in { ExternalAccessible := 'False'; ExternalVisible := 'False'; ExternalWritable := 'False'} : Int;   // PIW to be unscaled
      generalackn { ExternalAccessible := 'False'; ExternalVisible := 'False'; ExternalWritable := 'False'} : Bool;   // General acknowledgement
      reset { ExternalAccessible := 'False'; ExternalVisible := 'False'; ExternalWritable := 'False'} : Bool;   // Reset faults
      mute { ExternalAccessible := 'False'; ExternalVisible := 'False'; ExternalWritable := 'False'} : Bool;   // Mute siren
      p1s { ExternalAccessible := 'False'; ExternalVisible := 'False'; ExternalWritable := 'False'} : Bool;   // Pulse edge for 1Hz
      p100ms { ExternalAccessible := 'False'; ExternalVisible := 'False'; ExternalWritable := 'False'} : Bool;   // Pulse edge for 10Hz
      t_sys {InstructionName := 'DTL'; LibVersion := '1.0'; ExternalAccessible := 'False'; ExternalVisible := 'False'; ExternalWritable := 'False'} : DTL;   // System time
      "type" { ExternalAccessible := 'False'; ExternalVisible := 'False'; ExternalWritable := 'False'} : UInt;   // Type of measurement: 0=hmi, 1=H-L, 2=factor
   END_VAR

   VAR_OUTPUT 
      output { ExternalAccessible := 'False'; ExternalVisible := 'False'; ExternalWritable := 'False'} : Real;   // Scaled Value
   END_VAR

   VAR_IN_OUT 
      faults : "UDT_AINFAULTS";   // External data (Primary fault data - alarm & plc ackn)
      warnings : "UDT_AINWARNS";   // External data (Primary warning data - alarm & plc ackn)
   END_VAR

   VAR DB_SPECIFIC
      i : "UDT_AIN";   // UDT containing scale process data
   END_VAR
   VAR 
      exp { ExternalAccessible := 'False'; ExternalVisible := 'False'; ExternalWritable := 'False'} : Struct   // Exponential smoothing operands
         init { ExternalAccessible := 'False'; ExternalVisible := 'False'; ExternalWritable := 'False'} : Bool;   // Initialization routine
         Sn { ExternalAccessible := 'False'; ExternalVisible := 'False'; ExternalWritable := 'False'} : Real;   // Sn = n - output of smoothing
         Xn { ExternalAccessible := 'False'; ExternalVisible := 'False'; ExternalWritable := 'False'} : Real;   // Xn = n - sample of analog value
         lim_up { ExternalAccessible := 'False'; ExternalVisible := 'False'; ExternalWritable := 'False'} : Real;   // Limit up
         lim_down { ExternalAccessible := 'False'; ExternalVisible := 'False'; ExternalWritable := 'False'} : Real;   // Limit down
         t_buf {InstructionName := 'DTL'; LibVersion := '1.0'; ExternalAccessible := 'False'; ExternalVisible := 'False'; ExternalWritable := 'False'} : DTL;   // Time buffering from last call of the function
         t_diff { ExternalAccessible := 'False'; ExternalVisible := 'False'; ExternalWritable := 'False'} : Bool;   // t_diff = t_sys - t_buf (Ltime, ns)
      END_STRUCT;
      calc { ExternalAccessible := 'False'; ExternalVisible := 'False'; ExternalWritable := 'False'} : Struct   // Calculations for scaling process
         scalespan { ExternalAccessible := 'False'; ExternalVisible := 'False'; ExternalWritable := 'False'} : Real;   // Scaling span
         chnspan { ExternalAccessible := 'False'; ExternalVisible := 'False'; ExternalWritable := 'False'} : Real;   // Channel span
         xmax { ExternalAccessible := 'False'; ExternalVisible := 'False'; ExternalWritable := 'False'} : Real;   // Channel maximum value
         xmin { ExternalAccessible := 'False'; ExternalVisible := 'False'; ExternalWritable := 'False'} : Real;   // Channel minimum value
         ymax { ExternalAccessible := 'False'; ExternalVisible := 'False'; ExternalWritable := 'False'} : Real;   // Output maximum value
         ymin { ExternalAccessible := 'False'; ExternalVisible := 'False'; ExternalWritable := 'False'} : Real;   // Output minimum value
         x { ExternalAccessible := 'False'; ExternalVisible := 'False'; ExternalWritable := 'False'} : Real;   // Active x value (channel)
         y { ExternalAccessible := 'False'; ExternalVisible := 'False'; ExternalWritable := 'False'} : Real;   // Active y value (output)
         sign { ExternalAccessible := 'False'; ExternalVisible := 'False'; ExternalWritable := 'False'} : Bool;   // Linear scaling slope sign
         scale { ExternalAccessible := 'False'; ExternalVisible := 'False'; ExternalWritable := 'False'} : Struct   // Scaling
            "type" { ExternalAccessible := 'False'; ExternalVisible := 'False'; ExternalWritable := 'False'; S7_SetPoint := 'True'} : UInt;   // Type of measurement: 0=hmi, 1=H-L, 2=factor
            in { ExternalAccessible := 'False'; ExternalVisible := 'False'; ExternalWritable := 'False'} : Real;   // Input to real number
            scalehigh { ExternalAccessible := 'False'; ExternalVisible := 'False'; ExternalWritable := 'False'; S7_SetPoint := 'True'} : Real;   // High limit of scale process
            scalelow { ExternalAccessible := 'False'; ExternalVisible := 'False'; ExternalWritable := 'False'; S7_SetPoint := 'True'} : Real;   // Low limit of scale process
            channelhigh { ExternalAccessible := 'False'; ExternalVisible := 'False'; ExternalWritable := 'False'; S7_SetPoint := 'True'} : Real;   // Channel high limit (ex. 27648)
            channellow { ExternalAccessible := 'False'; ExternalVisible := 'False'; ExternalWritable := 'False'; S7_SetPoint := 'True'} : Real;   // Channel high limit (ex. 0)
            factor { ExternalAccessible := 'False'; ExternalVisible := 'False'; ExternalWritable := 'False'; S7_SetPoint := 'True'} : Real;   // Factor multiplied to real number
            calc1 { ExternalAccessible := 'False'; ExternalVisible := 'False'; ExternalWritable := 'False'} : Real;   // Calculation intermediate
            span { ExternalAccessible := 'False'; ExternalVisible := 'False'; ExternalWritable := 'False'} : Real;   // Span value
            output { ExternalAccessible := 'False'; ExternalVisible := 'False'; ExternalWritable := 'False'} : Real;   // Scaled value
         END_STRUCT;
      END_STRUCT;
      lastob_si {InstructionName := 'SI_classic'; LibVersion := '1.0'; ExternalAccessible := 'False'; ExternalVisible := 'False'; ExternalWritable := 'False'; S7_SetPoint := 'False'} : SI_classic;   // System info type (Last OB call info)
      startob_si {InstructionName := 'SI_classic'; LibVersion := '1.0'; ExternalAccessible := 'False'; ExternalVisible := 'False'; ExternalWritable := 'False'; S7_SetPoint := 'False'} : SI_classic;   // System info type (Startup OB call info)
      err { ExternalAccessible := 'False'; ExternalVisible := 'False'; ExternalWritable := 'False'} : Int;   // System info retval
      hilow { ExternalAccessible := 'False'; ExternalVisible := 'False'; ExternalWritable := 'False'} : Bool;   // Scaling based on hi-low
      factor { ExternalAccessible := 'False'; ExternalVisible := 'False'; ExternalWritable := 'False'} : Bool;   // Scaling based on factor
   END_VAR


BEGIN
	REGION GEN  NW:2-3
	    
	    //Network2: GEN: Move FC Inputs to UDT Inputs
	    
	    // IF #type = 1 OR #type = 2 THEN
	    //     #i.chn.type := #type;
	    // END_IF;
	    
	    //Network3: AIN: Convert analog input (AIN) to real
	    
	    #i.chn.in := INT_TO_REAL(#in);
	    
	END_REGION
	
	REGION SCALE  NW:4-7
	    
	    //Network4: AIN: Crosscheck if scaling is complete
	    
	    #hilow := #i.chn.type = 1 AND #i.scale.high <> #i.scale.low AND #i.chn.high <> #i.chn.low;
	    #factor := #i.chn.type = 2 AND #i.scale.factor <> 0.0;
	    
	    #i.scale.set := #hilow OR #factor;
	    
	    //Network5: AIN: Determine sign of scaling slope and calculation operands (Hi - Low)
	    
	    IF #i.scale.set AND #hilow THEN
	        #calc.scalespan := #i.scale.high - #i.scale.low;
	        #calc.chnspan := #i.chn.high - #i.chn.low;
	        #calc.x := #i.chn.in;
	        IF #calc.scalespan > 0 AND #calc.chnspan > 0 THEN
	            #calc.sign := TRUE;
	            #calc.ymax := #i.scale.high;
	            #calc.ymin := #i.scale.low;
	            #calc.xmax := #i.chn.high;
	            #calc.xmin := #i.chn.low;
	        ELSIF #calc.scalespan < 0 AND #calc.chnspan < 0 THEN
	            #calc.sign := TRUE;
	            #calc.ymax := #i.scale.low;
	            #calc.ymin := #i.scale.high;
	            #calc.xmax := #i.chn.low;
	            #calc.xmin := #i.chn.high;
	        ELSIF #calc.scalespan < 0 AND #calc.chnspan > 0 THEN
	            #calc.sign := FALSE;
	            #calc.ymax := #i.scale.low;
	            #calc.ymin := #i.scale.high;
	            #calc.xmax := #i.chn.high;
	            #calc.xmin := #i.chn.low;
	        ELSE
	            #calc.sign := FALSE;
	            #calc.ymax := #i.scale.high;
	            #calc.ymin := #i.scale.low;
	            #calc.xmax := #i.chn.low;
	            #calc.xmin := #i.chn.high;
	        END_IF;
	    ELSE
	        #calc.scalespan := #calc.chnspan := #calc.xmax := #calc.xmin := #calc.ymax := #calc.ymin := 0;
	    END_IF;
	    
	    //Network6: AIN: Determine sign of scaling slope and calculation operands (Hi - Low)
	    
	    IF #hilow AND #calc.sign THEN
	        
	        #calc.y := #calc.ymin + ((#calc.ymax - #calc.ymin) * (#calc.x - #calc.xmin) / (#calc.xmax - #calc.xmin));
	        
	        IF #calc.x <= #calc.xmin THEN
	            #calc.y := #calc.ymin;
	        END_IF;
	        
	        IF #calc.x >= #calc.xmax THEN
	            #calc.y := #calc.ymax;
	        END_IF;
	        
	    END_IF;
	    
	    IF #hilow AND NOT #calc.sign THEN
	        
	        #calc.y := #calc.ymin + ((#calc.ymax - #calc.ymin) * (#calc.xmax - #calc.x) / (#calc.xmax - #calc.xmin));
	        
	        IF #calc.x <= #calc.xmin THEN
	            #calc.y := #calc.ymax;
	        END_IF;
	        
	        IF #calc.x >= #calc.xmax THEN
	            #calc.y := #calc.ymin;
	        END_IF;
	        
	    END_IF;
	    
	    IF #hilow THEN
	        #i.scaled := #calc.y;
	    END_IF;
	    
	    //Network7: AIN: Scale AIN (Factor)
	    
	    IF #factor THEN
	        #i.scaled := #i.chn.in * #i.scale.factor;
	    END_IF;
	    
	    IF #factor AND #i.chn.in <= -32768.0 THEN
	        #i.scaled := -9999.0;
	    END_IF;
	    
	    IF #factor AND #i.chn.in >= 32767.0 THEN
	        #i.scaled := 9999.0;
	    END_IF;
	    
	END_REGION
	
	REGION SMOOTHING  NW:8
	    
	    //Network8: FILTER: Exponential smoothing
	    
	    IF #i.exp."en" AND NOT #i.sim."en" AND #i.scale.set AND FALSE THEN
	        
	        // Check system
	        #err := RD_SINFO(TOP_SI => #lastob_si, START_UP_SI => #startob_si);
	        
	        // Init routine
	        IF #lastob_si.EV_NUM = 1 OR #lastob_si.EV_NUM = 2 OR #lastob_si.EV_NUM = 4 THEN
	            #exp.init := false;
	        END_IF;
	        
	        // Enter routine
	        #exp.Xn := #i.scaled;
	        #exp.lim_up := #exp.Xn + #i.exp.limit;
	        #exp.lim_down := #exp.Xn - #i.exp.limit;
	        
	        //#exp.t_diff := T_DIFF(IN1 := #t_sys, IN2 := #exp.t_buf);
	        //#i.exp.dt := UDINT_TO_REAL(LTIME_TO_UDINT(#exp.t_diff)) / 1000000.0;
	        
	        IF #i.exp.T <= 0 THEN // Force the period to be higher than 0 to avoid infinity on the exponent
	            #i.exp.T := #i.exp.dt / 1000.0;
	        END_IF;
	        
	        IF #i.exp.dt > 0 AND #i.exp.T > #i.exp.dt / 1000.0 THEN
	            #i.exp.a := 1 - EXP(- #i.exp.dt / (1000.0 * #i.exp.T));
	        END_IF;
	        
	(* startup initialisation *)
	        IF NOT #exp.init OR #i.exp.a <= 0 OR #i.exp.a >= 1 THEN
	            #exp.init := TRUE;
	            #exp.Sn := #exp.Xn;
	        ELSIF #exp.Sn >= #exp.lim_down AND #exp.Sn <= #exp.lim_up THEN
	            #exp.Sn := #exp.Xn;
	        ELSE
	            #exp.Sn := #exp.Sn + (#exp.Xn - #exp.Sn) * #i.exp.a;
	        END_IF;
	        
	    ELSE
	        #exp.init := false;
	        #exp.Xn := #i.scaled;
	        #exp.Sn := #i.scaled;
	        
	    END_IF;
	    
	    // Buffering
	    #exp.t_buf := #t_sys;
	    
	    // Output
	    #i.exp.init := #exp.init;
	    #i.output := #exp.Sn;
	    
	END_REGION
	
	REGION SIMULATION  NW:9
	    
	    //Network9: SIM: Simulation
	    
	    IF #i.sim."en" THEN
	        #i.output := #i.sim.value;
	    END_IF;
	    
	END_REGION
	
	REGION FAULTS  NW:10-13
	    
	    //Network10: FAULT: HH
	    
	    "AFC_AlarmAckn"(trigger := #i.output >= #i.faults.sp_hh,
	                    release := TRUE,
	                    ctrlpoint := FALSE,
	                    enackn := TRUE,
	                    ensiren := TRUE,
	                    p100ms := #p100ms,
	                    generalackn := #generalackn OR #i.faults.fpreset,
	                    reset := #reset OR #i.faults.fpreset,
	                    mute := #mute,
	                    delay := 0.0,
	                    plcackn => #faults.ctrl.plcackn_hh,
	                    alarm => #faults.ctrl.alarm_hh,
	                    siren => #faults.status.siren_hh,
	                    hmiackn := #faults.status.hmiackn_hh,
	                    Data := #i.faults.hh);
	    
	    //Network11: FAULT: LL
	    
	    "AFC_AlarmAckn"(trigger := #i.output <= #i.faults.sp_ll,
	                    release := TRUE,
	                    ctrlpoint := FALSE,
	                    enackn := TRUE,
	                    ensiren := TRUE,
	                    p100ms := #p100ms,
	                    generalackn := #generalackn OR #i.faults.fpreset,
	                    reset := #reset OR #i.faults.fpreset,
	                    mute := #mute,
	                    delay := 0.0,
	                    plcackn => #faults.ctrl.plcackn_ll,
	                    alarm => #faults.ctrl.alarm_ll,
	                    siren => #faults.status.siren_ll,
	                    hmiackn := #faults.status.hmiackn_ll,
	                    Data := #i.faults.ll);
	    
	    //Network12: WARNING: H
	    
	    "AFC_AlarmAckn"(trigger := #i.output >= #i.faults.sp_h,
	                    release := TRUE,
	                    ctrlpoint := FALSE,
	                    enackn := TRUE,
	                    ensiren := TRUE,
	                    p100ms := #p100ms,
	                    generalackn := #generalackn OR #i.faults.fpreset,
	                    reset := #reset OR #i.faults.fpreset,
	                    mute := #mute,
	                    delay := 0.0,
	                    plcackn => #warnings.ctrl.plcackn_h,
	                    alarm => #warnings.ctrl.alarm_h,
	                    siren => #warnings.status.siren_h,
	                    hmiackn := #warnings.status.hmiackn_h,
	                    Data := #i.faults.h);
	    
	    //Network13: WARNING: L
	    
	    "AFC_AlarmAckn"(trigger := #i.output <= #i.faults.sp_l,
	                    release := TRUE,
	                    ctrlpoint := FALSE,
	                    enackn := TRUE,
	                    ensiren := TRUE,
	                    p100ms := #p100ms,
	                    generalackn := #generalackn OR #i.faults.fpreset,
	                    reset := #reset OR #i.faults.fpreset,
	                    mute := #mute,
	                    delay := 0.0,
	                    plcackn => #warnings.ctrl.plcackn_l,
	                    alarm => #warnings.ctrl.alarm_l,
	                    siren => #warnings.status.siren_l,
	                    hmiackn := #warnings.status.hmiackn_l,
	                    Data := #i.faults.l);
	    
	END_REGION
	
	REGION TREND  NW:14-15
	    
	    //Network14: TREND: Set trend high - low limit
	    
	    IF #hilow THEN
	        #i.trendhigh := #calc.ymax + ABS(#calc.ymax) * 0.1;
	        #i.trendlow := #calc.ymin - ABS(#calc.ymax) * 0.1;
	    END_IF;
	    
	    //Network15: TREND: Set trend high - low limit
	    
	    IF #hilow THEN
	        #i.trendhigh := 1.2 * #i.scale.low;
	    END_IF;
	    
	    IF #hilow THEN
	        #i.trendhigh := 1.2 * #i.scale.high;
	    END_IF;
	    
	END_REGION
	
	REGION OUTPUT  NW:16
	    
	    //Network16: OUTPUT: Write to output
	#output := #i.output;
	    
	END_REGION
	
	REGION BUTTON  NW:17
	    
	    //Network17: EXTRA: Button treatment
	    
	    IF #i.faults.fpreset THEN
	        #i.faults.fpreset := FALSE;
	    END_IF;
	    
	END_REGION
END_FUNCTION_BLOCK

FUNCTION_BLOCK "AFB_ControlValve_v3"
{ S7_Optimized_Access := 'TRUE' }
VERSION : 0.1
   VAR_INPUT 
      control { ExternalAccessible := 'False'; ExternalVisible := 'False'; ExternalWritable := 'False'} : Bool;   // Request for auto control
      spsource { ExternalAccessible := 'False'; ExternalVisible := 'False'; ExternalWritable := 'False'} : Bool;   // 0=internal setpoint, 1=external setpoint
      followup { ExternalAccessible := 'False'; ExternalVisible := 'False'; ExternalWritable := 'False'} : Bool;   // 0=motor control from PID, 1=motor setpoint directly from program
      pidrun { ExternalAccessible := 'False'; ExternalVisible := 'False'; ExternalWritable := 'False'} : Bool;   // 0=controller not ready, controller is running
      block { ExternalAccessible := 'False'; ExternalVisible := 'False'; ExternalWritable := 'False'} : Bool;   // Block control of valve
      p1s { ExternalAccessible := 'False'; ExternalVisible := 'False'; ExternalWritable := 'False'} : Bool;   // Pulse that is generated every 1 sec
      p100ms { ExternalAccessible := 'False'; ExternalVisible := 'False'; ExternalWritable := 'False'} : Bool;   // Pulse that is generated every 100 msec
      blink { ExternalAccessible := 'False'; ExternalVisible := 'False'; ExternalWritable := 'False'} : Bool;   // Blink that is used for the graphics
      PV { ExternalAccessible := 'False'; ExternalVisible := 'False'; ExternalWritable := 'False'} : Real;   // Reference for PID
      PV_unit { ExternalAccessible := 'False'; ExternalVisible := 'False'; ExternalWritable := 'False'} : WString;   // Peripheral value unit
      EXT_SP { ExternalAccessible := 'False'; ExternalVisible := 'False'; ExternalWritable := 'False'} : Real;   // External setpoint
      FUP { ExternalAccessible := 'False'; ExternalVisible := 'False'; ExternalWritable := 'False'} : Real;   // Follow up value
      Out_unit { ExternalAccessible := 'False'; ExternalVisible := 'False'; ExternalWritable := 'False'} : WString;   // Output unit (If nothing is entered then it is from the HMI)
   END_VAR

   VAR_OUTPUT 
      reference { ExternalAccessible := 'False'; ExternalVisible := 'False'; ExternalWritable := 'False'} : Int;   // Valve reference
   END_VAR

   VAR RETAIN
      i : "UDT_CONTROLVALVE";   // UDT containing control valve data
   END_VAR
   VAR 
      cont { ExternalAccessible := 'False'; ExternalVisible := 'False'; ExternalWritable := 'False'} : Struct   // Controller
         COM_RST { ExternalAccessible := 'False'; ExternalVisible := 'False'; ExternalWritable := 'False'} : Bool;   // Restart command
         MAN_ON { ExternalAccessible := 'False'; ExternalVisible := 'False'; ExternalWritable := 'False'} : Bool;   // Manual control
         SP_INT { ExternalAccessible := 'False'; ExternalVisible := 'False'; ExternalWritable := 'False'} : Real;   // Setpoint internal
         PV_IN { ExternalAccessible := 'False'; ExternalVisible := 'False'; ExternalWritable := 'False'} : Real;   // Peripheral value
         GAIN { ExternalAccessible := 'False'; ExternalVisible := 'False'; ExternalWritable := 'False'} : Real;   // Proportional gain loaded according to the action (signed)
         TI { ExternalAccessible := 'False'; ExternalVisible := 'False'; ExternalWritable := 'False'} : Time;   // Integral time
         TD { ExternalAccessible := 'False'; ExternalVisible := 'False'; ExternalWritable := 'False'} : Time;   // Derivative time
         LMN_HLM { ExternalAccessible := 'False'; ExternalVisible := 'False'; ExternalWritable := 'False'} : Real;   // Controller's higher LMN value (%)
         LMN_LLM { ExternalAccessible := 'False'; ExternalVisible := 'False'; ExternalWritable := 'False'} : Real;   // Controller's lower LMN value (%)
         LMN_FAC { ExternalAccessible := 'False'; ExternalVisible := 'False'; ExternalWritable := 'False'} : Real;   // LMN factor
         LMN_OFF { ExternalAccessible := 'False'; ExternalVisible := 'False'; ExternalWritable := 'False'} : Real;   // LMN offset
         I_ITLVAL { ExternalAccessible := 'False'; ExternalVisible := 'False'; ExternalWritable := 'False'} : Real;   // Controller's integral initialization value (%)
         LMN { ExternalAccessible := 'False'; ExternalVisible := 'False'; ExternalWritable := 'False'} : Real;   // Controller's manipulated value
      END_STRUCT;
      calc { ExternalAccessible := 'False'; ExternalVisible := 'False'; ExternalWritable := 'False'} : Struct   // Calculations for scaling process
         inspan { ExternalAccessible := 'False'; ExternalVisible := 'False'; ExternalWritable := 'False'} : Real;   // Scaling span
         outspan { ExternalAccessible := 'False'; ExternalVisible := 'False'; ExternalWritable := 'False'} : Real;   // Channel span
         xmax { ExternalAccessible := 'False'; ExternalVisible := 'False'; ExternalWritable := 'False'} : Real;   // Channel maximum value
         xmin { ExternalAccessible := 'False'; ExternalVisible := 'False'; ExternalWritable := 'False'} : Real;   // Channel minimum value
         ymax { ExternalAccessible := 'False'; ExternalVisible := 'False'; ExternalWritable := 'False'} : Real;   // Output maximum value
         ymin { ExternalAccessible := 'False'; ExternalVisible := 'False'; ExternalWritable := 'False'} : Real;   // Output minimum value
         x { ExternalAccessible := 'False'; ExternalVisible := 'False'; ExternalWritable := 'False'} : Real;   // Active x value (channel)
         y { ExternalAccessible := 'False'; ExternalVisible := 'False'; ExternalWritable := 'False'} : Real;   // Active y value (output)
         sign { ExternalAccessible := 'False'; ExternalVisible := 'False'; ExternalWritable := 'False'} : Bool;   // Linear scaling slope sign
      END_STRUCT;
   END_VAR

   VAR_TEMP 
      condSET : Bool;
      condRESET : Bool;
   END_VAR


BEGIN
	REGION GEN  NW:2
	    
	    //Network2: GEN: Move FC inputs to UDT inputs
	    
	    #i.pid.spsource := #spsource;
	    #i.pid.followup := #followup;
	    #i.pid.pidrun := #pidrun;
	    #i.pid.PV := #PV;
	    #i.pid.EXT_SP := #EXT_SP;
	    #i.pid.FUP := #FUP;
	    #i.pid.pvunit := #PV_unit;
	    
	    IF #Out_unit <> WSTRING#'' THEN
	        #i.pid.outunit := #Out_unit;
	    END_IF;
	    
	END_REGION
	
	REGION STATUS  NW:3
	    
	    //Network3: STATUS: Start interlock
	    
	    #i.status.ilstart := NOT #block AND #i.unscale.set;
	    
	END_REGION
	
	REGION FEEDBACK  NW:4-5
	    
	    //Network4: FEEDBACK: Virtual feedback "Open"
	    
	    #i.out.vfbact := #i.pid.OP > #i.unscale.inlow;
	    
	    //Network5: FEEDBACK: Virtual feedback "Close"
	    
	    #i.out.vfbdeact := #i.pid.OP <= #i.unscale.inlow;
	    
	END_REGION
	
	REGION OUTPUT  NW:6
	    
	    //Network6: OUTPUT: Enable control of valve
	    
	    #i.out.control := #i.status.ilstart AND (#control OR #i.pid.mode);
	    
	END_REGION
	
	REGION LOAD PID  NW:7
	    
	    //Network7: CONTROLLER: Load from PID block
	    
	    #i.pid.LMN := #cont.LMN;
	    
	END_REGION
	
	REGION PID  NW:8-14
	    
	    //Network8: PID: Manage controller's limits
	    
	    IF #i.pid.H <= #i.pid.L THEN
	        #i.pid.H := #i.pid.L := #calc.xmin;
	    END_IF;
	    
	    IF #i.pid.H > #calc.xmax THEN
	        #i.pid.H := #calc.xmax;
	    END_IF;
	    
	    IF #i.pid.L < #calc.xmin THEN
	        #i.pid.L := #calc.xmin;
	    END_IF;
	    
	    IF (#i.pid.ITLVAL < #i.pid.L) AND (#i.pid.ITLVAL > #i.pid.H) THEN
	        #i.pid.ITLVAL := #calc.xmin;
	    END_IF;
	    
	    IF (#i.pid.OFFVAL < #i.pid.L) AND (#i.pid.ITLVAL > #i.pid.H) THEN
	        #i.pid.OFFVAL := #calc.xmin;
	    END_IF;
	    
	    //Network9: PID: Load SP
	    
	    IF #i.pid.spsource THEN
	        #i.pid.SP := #i.pid.EXT_SP;
	    END_IF;
	    
	    //Network10: PID: Determine if initialization routine is required
	    
	    #i.pid.init.req := (#i.pid.ITLVAL > #i.pid.L) AND (#i.pid.init.dur > 0.0);
	    
	    //Network11: PID: Determine the delay SP
	    
	    IF NOT #i.out.control AND #i.pid.init.req THEN
	        #i.pid.init.delay.in.spon := #i.pid.init.dur;
	    END_IF;
	    
	    IF NOT #i.out.control AND NOT #i.pid.init.req THEN
	        #i.pid.init.delay.in.spon := 0.0;
	    END_IF;
	    
	    IF #i.pid.mode = #i.pid.followup THEN
	        #i.pid.init.delay.in.spon := 0.0;
	    END_IF;
	    
	    //Network12: PID: Delay for holding an init value
	    
	    "AFC_DelayONOFF"(cmd := #i.out.control,
	                     Pulse := #p100ms,
	                     Reset := NOT #i.out.control,
	                     on => #i.pid.init.delay.out.on,
	                     Data := #i.pid.init.delay);
	    
	    //Network13: PID: Reset the controller
	    
	    #i.pid.cmdrst := NOT #i.pid.init.delay.out.on OR #i.pid.mode OR #i.pid.followup;
	    
	    //Network14: PID: Load output
	    
	    IF NOT #i.pid.mode THEN
	        
	        IF #i.out.control THEN
	            
	            IF NOT #i.pid.followup THEN
	                
	                IF #i.pid.pidrun THEN
	                    #i.pid.OP := #i.pid.LMN;
	                END_IF;
	                
	                IF #i.pid.cmdrst THEN
	                    #i.pid.OP := #i.pid.ITLVAL;
	                END_IF;
	                
	            END_IF;
	            
	        ELSIF #i.pid.followup THEN
	            
	            #i.pid.OP := #i.pid.FUP;
	            
	        END_IF;
	        
	    ELSIF #i.pid.mode THEN
	        
	        IF NOT #i.out.control THEN
	            #i.pid.OP := #i.pid.OFFVAL;
	        END_IF;
	        
	    END_IF;
	    
	END_REGION
	
	REGION UNSCALE  NW:15-19
	    
	    //Network15: UNSCALE: Move input
	    
	    #i.unscale.in := #i.pid.OP;
	    
	    //Network16: UNSCALE: Cross-check unscaling setup
	    
	    #i.unscale.set := (#i.unscale.inhigh <> #i.unscale.inlow) AND (#i.unscale.outhigh <> #i.unscale.inlow);
	    
	    //Network17: UNSCALE: Determine sign of scaling slope and calculation operands (Hi - Low)
	    
	    IF #i.unscale.set THEN
	        #calc.inspan := #i.unscale.inhigh - #i.unscale.inlow;
	        #calc.outspan := #i.unscale.outhigh - #i.unscale.outlow;
	        #calc.x := #i.unscale.in;
	        IF #calc.inspan > 0 AND #calc.outspan > 0 THEN
	            #calc.sign := TRUE;
	            #calc.ymax := #i.unscale.outhigh;
	            #calc.ymin := #i.unscale.outlow;
	            #calc.xmax := #i.unscale.inhigh;
	            #calc.xmin := #i.unscale.inlow;
	        ELSIF #calc.inspan < 0 AND #calc.outspan < 0 THEN
	            #calc.sign := TRUE;
	            #calc.ymax := #i.unscale.outlow;
	            #calc.ymin := #i.unscale.outhigh;
	            #calc.xmax := #i.unscale.inlow;
	            #calc.xmin := #i.unscale.inhigh;
	        ELSIF #calc.inspan < 0 AND #calc.outspan > 0 THEN
	            #calc.sign := FALSE;
	            #calc.ymax := #i.unscale.outlow;
	            #calc.ymin := #i.unscale.outhigh;
	            #calc.xmax := #i.unscale.inhigh;
	            #calc.xmin := #i.unscale.inlow;
	        ELSE
	            #calc.sign := FALSE;
	            #calc.ymax := #i.unscale.outhigh;
	            #calc.ymin := #i.unscale.outlow;
	            #calc.xmax := #i.unscale.inlow;
	            #calc.xmin := #i.unscale.inhigh;
	        END_IF;
	    ELSE
	        #calc.inspan := #calc.outspan := #calc.xmax := #calc.xmin := #calc.ymax := #calc.ymin := 0;
	    END_IF;
	    
	    //Network18: UNSCALE: Determine output
	    
	    IF #i.unscale.set AND #calc.sign THEN
	        
	        #calc.y := #calc.ymin + ((#calc.ymax - #calc.ymin) * (#calc.x - #calc.xmin) / (#calc.xmax - #calc.xmin));
	        
	        IF #calc.x <= #calc.xmin THEN
	            #calc.y := #calc.ymin;
	        END_IF;
	        
	        IF #calc.x >= #calc.xmax THEN
	            #calc.y := #calc.ymax;
	        END_IF;
	        
	    END_IF;
	    
	    IF #i.unscale.set AND NOT #calc.sign THEN
	        
	        #calc.y := #calc.ymin + ((#calc.ymax - #calc.ymin) * (#calc.xmax - #calc.x) / (#calc.xmax - #calc.xmin));
	        
	        IF #calc.x <= #calc.xmin THEN
	            #calc.y := #calc.ymax;
	        END_IF;
	        
	        IF #calc.x >= #calc.xmax THEN
	            #calc.y := #calc.ymin;
	        END_IF;
	        
	    END_IF;
	    
	    IF #i.unscale.set THEN
	        #i.unscale.output := #calc.y;
	    END_IF;
	    
	    IF NOT #i.unscale.set THEN
	        #i.unscale.output := 0.0;
	    END_IF;
	    
	    //Network19: UNSCALE: Convert to INT
	    
	    #i.out."ref" := REAL_TO_INT(#i.unscale.output);
	    
	    
	END_REGION
	
	REGION LOAD PID  NW:20
	    
	    //Network20: CONTROLLER: Load to PID block
	    
	    #cont.COM_RST := #i.pid.cmdrst;
	    
	    #cont.MAN_ON := #i.pid.mode;
	    
	    #cont.SP_INT := #i.pid.SP;
	    
	    #cont.PV_IN := #i.pid.PV;
	    
	    IF #i.pid.action THEN
	        #cont.GAIN := ABS_REAL(#i.pid.P);
	    ELSE
	        #cont.GAIN := 0.0 - ABS_REAL(#i.pid.P);
	    END_IF;
	    
	    #cont.TI := DINT_TO_TIME(#i.pid.I);
	    
	    #cont.TD := DINT_TO_TIME(#i.pid.D);
	    
	    #cont.LMN_HLM := ((#i.pid.H - #calc.xmin) / (#calc.xmax - #calc.xmin)) * 100.0;
	    
	    #cont.LMN_LLM := ((#i.pid.L - #calc.xmin) / (#calc.xmax - #calc.xmin)) * 100.0;
	    
	    #cont.LMN_FAC := (#calc.xmax - #calc.xmin) / 100.0;
	    
	    #cont.LMN_OFF := #calc.xmin;
	    
	    #cont.I_ITLVAL := ((#i.pid.OP - #calc.xmin) / (#calc.xmax - #calc.xmin)) * 100.0;
	    
	END_REGION
	
	REGION STATUS  NW:21
	    
	    //Network21: STATUS: Icon
	    
	    #i.status.icon := 0;
	    
	    IF #i.out.vfbact
	    THEN
	        #i.status.icon := 1;
	    ELSIF FALSE AND #blink
	    THEN
	        #i.status.icon := 3;
	    END_IF;
	    
	END_REGION
	
	REGION OUTPUT  NW:22
	    
	    //Network22: OUTPUT: Move to FC outputs
	    
	    #reference := #i.out."ref";
	    
	END_REGION
END_FUNCTION_BLOCK

FUNCTION_BLOCK "AFB_DIFF_v3"
{ S7_Optimized_Access := 'TRUE' }
VERSION : 0.1
   VAR_INPUT 
      Minuend { ExternalAccessible := 'False'; ExternalVisible := 'False'; ExternalWritable := 'False'} : Real;   // Minuend of subtraction
      Subtrahend { ExternalAccessible := 'False'; ExternalVisible := 'False'; ExternalWritable := 'False'} : Real;   // Subtrahend of subtraction
      unit { ExternalAccessible := 'False'; ExternalVisible := 'False'; ExternalWritable := 'False'} : WString;   // Unit
      generalackn { ExternalAccessible := 'False'; ExternalVisible := 'False'; ExternalWritable := 'False'} : Bool;   // General acknowledgement
      reset { ExternalAccessible := 'False'; ExternalVisible := 'False'; ExternalWritable := 'False'} : Bool;   // Reset alarms
      mute { ExternalAccessible := 'False'; ExternalVisible := 'False'; ExternalWritable := 'False'} : Bool;   // Mute siren
      p1s { ExternalAccessible := 'False'; ExternalVisible := 'False'; ExternalWritable := 'False'} : Bool;   // Pulse edge for 1Hz
      p100ms { ExternalAccessible := 'False'; ExternalVisible := 'False'; ExternalWritable := 'False'} : Bool;   // Pulse edge for 10Hz
   END_VAR

   VAR_OUTPUT 
      output { ExternalAccessible := 'False'; ExternalVisible := 'False'; ExternalWritable := 'False'} : Real;   // Scaled Value
   END_VAR

   VAR_IN_OUT 
      faults : "UDT_AINFAULTS";   // External data (Primary fault data - alarm & plc ackn)
      warnings : "UDT_AINWARNS";   // External data (Primary warning data - alarm & plc ackn)
   END_VAR

   VAR RETAIN
      i : "UDT_DIFF";   // UDT containing scale process data
   END_VAR


BEGIN
	REGION GEN  NW:2
	    
	    //Network2: GEN: Move FC Inputs to UDT
	    
	    #i.minuend := #Minuend;
	    #i.subtrahend := #Subtrahend;
	    
	END_REGION
	
	REGION DIFF  NW:3-4
	    
	    //Network3: DIFF: Calculate Differential
	    
	    #i.output := #i.minuend - #i.subtrahend;
	    
	    //Network4: DIFF: Set unit
	    
	    #i.unit := #unit;
	    
	END_REGION
	
	REGION SIM  NW:5
	    
	    //Network5: SIM: Simulation
	    
	    IF #i.sim."en" THEN
	        #i.output := #i.sim.value;
	    END_IF;
	    
	END_REGION
	
	REGION FAULT  NW:6-9
	    
	    //Network6: FAULT: HH
	    
	    "AFC_AlarmAckn"(trigger := #i.output >= #i.faults.sp_hh,
	                    release := TRUE,
	                    ctrlpoint := FALSE,
	                    enackn := TRUE,
	                    ensiren := TRUE,
	                    p100ms := #p100ms,
	                    generalackn := #generalackn OR #i.faults.fpreset,
	                    reset := #reset OR #i.faults.fpreset,
	                    mute := #mute,
	                    delay := 0.0,
	                    plcackn => #faults.ctrl.plcackn_hh,
	                    alarm => #faults.ctrl.alarm_hh,
	                    siren => #faults.status.siren_hh,
	                    hmiackn := #faults.status.hmiackn_hh,
	                    Data := #i.faults.hh);
	    
	    //Network7: FAULT: LL
	    
	    "AFC_AlarmAckn"(trigger := #i.output <= #i.faults.sp_ll,
	                    release := TRUE,
	                    ctrlpoint := FALSE,
	                    enackn := TRUE,
	                    ensiren := TRUE,
	                    p100ms := #p100ms,
	                    generalackn := #generalackn OR #i.faults.fpreset,
	                    reset := #reset OR #i.faults.fpreset,
	                    mute := #mute,
	                    delay := 0.0,
	                    plcackn => #faults.ctrl.plcackn_ll,
	                    alarm => #faults.ctrl.alarm_ll,
	                    siren => #faults.status.siren_ll,
	                    hmiackn := #faults.status.hmiackn_ll,
	                    Data := #i.faults.ll);
	    
	    //Network8: WARNING: H
	    
	    "AFC_AlarmAckn"(trigger := #i.output >= #i.faults.sp_h,
	                    release := TRUE,
	                    ctrlpoint := FALSE,
	                    enackn := TRUE,
	                    ensiren := TRUE,
	                    p100ms := #p100ms,
	                    generalackn := #generalackn OR #i.faults.fpreset,
	                    reset := #reset OR #i.faults.fpreset,
	                    mute := #mute,
	                    delay := 0.0,
	                    plcackn => #warnings.ctrl.plcackn_h,
	                    alarm => #warnings.ctrl.alarm_h,
	                    siren => #warnings.status.siren_h,
	                    hmiackn := #warnings.status.hmiackn_h,
	                    Data := #i.faults.h);
	    
	    //Network9: WARNING: L
	    
	    "AFC_AlarmAckn"(trigger := #i.output <= #i.faults.sp_l,
	                    release := TRUE,
	                    ctrlpoint := FALSE,
	                    enackn := TRUE,
	                    ensiren := TRUE,
	                    p100ms := #p100ms,
	                    generalackn := #generalackn OR #i.faults.fpreset,
	                    reset := #reset OR #i.faults.fpreset,
	                    mute := #mute,
	                    delay := 0.0,
	                    plcackn => #warnings.ctrl.plcackn_l,
	                    alarm => #warnings.ctrl.alarm_l,
	                    siren => #warnings.status.siren_l,
	                    hmiackn := #warnings.status.hmiackn_l,
	                    Data := #i.faults.l);
	    
	END_REGION
	
	REGION OUTPUT  NW:10
	    
	    //Network10: OUTPUT: Write to output
	    
	    #output := #i.output;
	    
	END_REGION
	
	REGION BUTTON  NW:11
	    
	    //Network11: EXTRA: Button treatment
	    
	    IF #i.faults.fpreset THEN
	        #i.faults.fpreset := FALSE;
	    END_IF;
	    
	END_REGION
	
	
	
	
	
	
	
	
	
	
	
	
	
	
	
	
	
	
	
	
	
	
	
	
	
	
	
	
	
END_FUNCTION_BLOCK

FUNCTION_BLOCK "AFB_DIN_v3"
{ S7_Optimized_Access := 'TRUE' }
VERSION : 0.1
   VAR_INPUT 
      input { ExternalAccessible := 'False'; ExternalVisible := 'False'; ExternalWritable := 'False'} : Bool;   // Digital Switch input in normal state
      monitorfault { ExternalAccessible := 'False'; ExternalVisible := 'False'; ExternalWritable := 'False'} : Bool;   // Release fault monitoring
      p1s { ExternalAccessible := 'False'; ExternalVisible := 'False'; ExternalWritable := 'False'} : Bool;   // Pulse edge for 1Hz
      p100ms { ExternalAccessible := 'False'; ExternalVisible := 'False'; ExternalWritable := 'False'} : Bool;   // Pulse edge for 10Hz
      generalackn { ExternalAccessible := 'False'; ExternalVisible := 'False'; ExternalWritable := 'False'} : Bool;   // General acknowledgement
      reset { ExternalAccessible := 'False'; ExternalVisible := 'False'; ExternalWritable := 'False'} : Bool;   // Reset Fault
      mute { ExternalAccessible := 'False'; ExternalVisible := 'False'; ExternalWritable := 'False'} : Bool;   // Mute siren
   END_VAR

   VAR_OUTPUT 
      Switch { ExternalAccessible := 'False'; ExternalVisible := 'False'; ExternalWritable := 'False'} : Bool;   // Switch after time cross check
   END_VAR

   VAR_IN_OUT 
      alarm_din { ExternalAccessible := 'False'; ExternalVisible := 'False'; ExternalWritable := 'False'} : Bool;
      plcackn_din { ExternalAccessible := 'False'; ExternalVisible := 'False'; ExternalWritable := 'False'} : Bool;
      siren_din { ExternalAccessible := 'False'; ExternalVisible := 'False'; ExternalWritable := 'False'} : Bool;
      hmiackn_din { ExternalAccessible := 'False'; ExternalVisible := 'False'; ExternalWritable := 'False'} : Bool;
   END_VAR

   VAR RETAIN
      i : "UDT_DIN";   // Temporary Switch Data
   END_VAR

   VAR_TEMP 
      condSET : Bool;
      condRESET : Bool;
   END_VAR


BEGIN
	REGION SIM  NW:2-3
	    
	    //Network2: SIM: Simulation
	    
	    #i.sim.simulated := (#i.sim.simulated OR #i.sim.cmdon) AND NOT #i.sim.cmdoff;
	    
	    //Network3: SIM: Force
	    
	    #condSET := #i.sim.cmdforce;
	    #condRESET := #i.sim.cmdunforce OR NOT #i.sim.simulated;
	    
	    #i.sim.forced := (#i.sim.forced OR #condSET) AND NOT #condRESET;
	    
	END_REGION
	
	REGION STATUS  NW:4-6
	    
	    //Network4: STATUS: Raw input
	    
	    #i.status.rawinput := #input;
	    
	    //Network5: STATUS: Processed input 
	    
	    #i.status.processed := (#input AND NOT #i.setup.polarity) OR (NOT #input AND #i.setup.polarity);
	    
	    //Network6: STATUS: Alarm monitor 
	    
	    #i.status.alarm_monitor := #monitorfault AND #i.faults.din.setup."en";
	    
	END_REGION
	
	REGION DIN  NW:7-9
	    
	    //Network7: DIN: Reset actual timers 
	    
	    IF (#i.status.processed AND #i.status.switch_active) OR #i.sim.simulated THEN
	        #i."time".on_act := #i."time".off_act := 0;
	    END_IF;
	    
	    IF NOT (#i.status.processed OR #i.status.switch_active) OR #i.sim.simulated THEN
	        #i."time".on_act := #i."time".off_act := 0;
	    END_IF;
	    
	    //Network8: DIN: Counter
	    
	    IF #p1s AND (#i.status.processed AND NOT #i.status.switch_active) THEN
	        #i."time".on_act := #i."time".on_act + 1;
	    END_IF;
	    
	    IF #p1s AND (NOT #i.status.processed AND #i.status.switch_active) THEN
	        #i."time".off_act := #i."time".off_act + 1;
	    END_IF;
	    
	    //Network9: DIN: Set switch active
	    
	    #condSET := #i.sim.forced OR (#i.status.processed AND NOT #i.sim.simulated AND #i."time".on_act >= #i."time".on_set);
	    #condRESET := (NOT #i.sim.forced AND #i.sim.simulated) OR (NOT #i.status.processed AND NOT #i.sim.simulated AND #i."time".off_act >= #i."time".off_set);
	    
	    #i.status.switch_active := (#i.status.switch_active OR #condSET) AND NOT #condRESET;
	    
	END_REGION
	
	REGION FAULT   NW:10
	    
	    //Network10: FAULT: Switch activated
	    
	    #condSET := NOT (#i.setup.triggerversion OR #i.status.switch_active) OR (#i.setup.triggerversion AND #i.status.switch_active);
	    
	    "AFC_AlarmAckn"(trigger := #condSET,
	                    release := #monitorfault,
	                    ctrlpoint := FALSE,
	                    enackn := TRUE,
	                    ensiren := TRUE,
	                    p100ms := #p100ms,
	                    generalackn := #generalackn OR #i.faults.fpreset,
	                    reset := #reset OR #i.faults.fpreset,
	                    mute := #mute,
	                    delay := 0.0,
	                    plcackn => #plcackn_din,
	                    alarm => #alarm_din,
	                    siren => #siren_din,
	                    hmiackn := #hmiackn_din,
	                    Data := #i.faults.din);
	    
	END_REGION
	
	REGION OUTPUT   NW:11
	    
	    //Network11: GEN: Move UDT Outputs to FC Outputs
	    
	    #Switch := #i.status.switch_active;
	    
	END_REGION
	
	REGION BUTTON  NW:12
	    
	    //Network12: EXTRA: Button treatment
	    
	    IF #i.faults.fpreset THEN
	        #i.faults.fpreset := FALSE;
	    END_IF;
	    
	END_REGION
END_FUNCTION_BLOCK

FUNCTION_BLOCK "AFB_MotorDirect_v3"
{ S7_Optimized_Access := 'TRUE' }
VERSION : 0.1
   VAR_INPUT 
      start { ExternalAccessible := 'False'; ExternalVisible := 'False'; ExternalWritable := 'False'} : Bool;   // "Logic" in order to start
      "fb" { ExternalAccessible := 'False'; ExternalVisible := 'False'; ExternalWritable := 'False'} : Bool;   // Motor's running feedback (1=run, 0=stop)
      mcb { ExternalAccessible := 'False'; ExternalVisible := 'False'; ExternalWritable := 'False'} : Bool;   // Motor circuit breaker (1=ok, 0=fault)
      ctrl { ExternalAccessible := 'False'; ExternalVisible := 'False'; ExternalWritable := 'False'} : Bool;   // Control of motor (1=PLC, 0=Local)
      block { ExternalAccessible := 'False'; ExternalVisible := 'False'; ExternalWritable := 'False'} : Bool;   // Condition that blocks motor operation
      generalackn { ExternalAccessible := 'False'; ExternalVisible := 'False'; ExternalWritable := 'False'} : Bool;   // General acknowledgement
      reset { ExternalAccessible := 'False'; ExternalVisible := 'False'; ExternalWritable := 'False'} : Bool;   // Option that resets the faults
      mute { ExternalAccessible := 'False'; ExternalVisible := 'False'; ExternalWritable := 'False'} : Bool;   // Mute siren
      autoset { ExternalAccessible := 'False'; ExternalVisible := 'False'; ExternalWritable := 'False'} : Bool;   // Option that sets the motor to auto mode (Used for mass auto set)
      manualset { ExternalAccessible := 'False'; ExternalVisible := 'False'; ExternalWritable := 'False'} : Bool;   // Option that sets the motor to manual mode (Used for mass manual set)
      p1s { ExternalAccessible := 'False'; ExternalVisible := 'False'; ExternalWritable := 'False'} : Bool;   // Pulse that is generated every 1 s (Count up)
      p100ms { ExternalAccessible := 'False'; ExternalVisible := 'False'; ExternalWritable := 'False'} : Bool;   // Pulse that is generated every 100 ms (Count up)
      blink { ExternalAccessible := 'False'; ExternalVisible := 'False'; ExternalWritable := 'False'} : Bool;   // Blink that is used for the graphics (Frequency of CPU)
   END_VAR

   VAR_OUTPUT 
      run { ExternalAccessible := 'False'; ExternalVisible := 'False'; ExternalWritable := 'False'} : Bool;   // Command to start motor
      vfb { ExternalAccessible := 'False'; ExternalVisible := 'False'; ExternalWritable := 'False'} : Bool;   // Virtual feedback (used everywhere instead of digital fb)
   END_VAR

   VAR_IN_OUT 
      faults : "UDT_MTRFAULTS";   // External data (Primary alarm data - alarm & plc ackn)
   END_VAR

   VAR RETAIN
      i : "UDT_MOTORDIRECT";   // Data type containing the motor's data
   END_VAR

   VAR_TEMP 
      condSET : Bool;
      condRESET : Bool;
   END_VAR


BEGIN
	REGION STATUS  NW:2-3
	    
	    //Network2: STATUS: Virtual feedback
	    
	    #i.status.vfb := (#fb AND NOT #i.sim.fb) OR (#i.out.run AND #i.sim.fb);
	    
	    //Network3: STATUS: Virtual control
	    
	    #i.status.vctrl := #i.sim.ctrl OR (#ctrl AND NOT #i.sim.ctrl);
	    
	END_REGION
	
	REGION FAULT  NW:4-8
	    
	    //Network4: FAULT: Fail to run
	    
	    "AFC_AlarmAckn"(trigger := NOT #i.status.vfb AND #i.out.run AND #i.status.vctrl,
	                    release := NOT #i.sim.fb,
	                    ctrlpoint := FALSE,
	                    enackn := TRUE,
	                    ensiren := TRUE,
	                    p100ms := #p100ms,
	                    generalackn := #generalackn OR #i.faults.fpreset,
	                    reset := #reset OR #i.faults.fpreset,
	                    mute := #mute,
	                    delay := 0.0,
	                    plcackn => #faults.ctrl.plcackn_ftr,
	                    alarm => #faults.ctrl.alarm_ftr,
	                    siren => #faults.status.siren_ftr,
	                    hmiackn := #faults.status.hmiackn_ftr,
	                    Data := #i.faults.ftr);
	    
	    //Network5: FAULT: Fail to stop
	    
	    "AFC_AlarmAckn"(trigger := #i.status.vfb AND NOT #i.out.run AND #i.status.vctrl,
	                    release := NOT #i.sim.fb,
	                    ctrlpoint := FALSE,
	                    enackn := TRUE,
	                    ensiren := TRUE,
	                    p100ms := #p100ms,
	                    generalackn := #generalackn OR #i.faults.fpreset,
	                    reset := #reset OR #i.faults.fpreset,
	                    mute := #mute,
	                    delay := 0.0,
	                    plcackn => #faults.ctrl.plcackn_fts,
	                    alarm => #faults.ctrl.alarm_fts,
	                    siren => #faults.status.siren_fts,
	                    hmiackn := #faults.status.hmiackn_fts,
	                    Data := #i.faults.fts);
	    
	    //Network6: FAULT: Monor circuit breaker
	    
	    "AFC_AlarmAckn"(trigger := NOT #mcb,
	                    release := NOT #i.sim.fb,
	                    ctrlpoint := FALSE,
	                    enackn := TRUE,
	                    ensiren := TRUE,
	                    p100ms := #p100ms,
	                    generalackn := #generalackn OR #i.faults.fpreset,
	                    reset := #reset OR #i.faults.fpreset,
	                    mute := #mute,
	                    delay := 0.0,
	                    plcackn => #faults.ctrl.plcackn_mcb,
	                    alarm => #faults.ctrl.alarm_mcb,
	                    siren => #faults.status.siren_mcb,
	                    hmiackn := #faults.status.hmiackn_mcb,
	                    Data := #i.faults.mcb);
	    
	    //Network7: FAULT: Control
	    
	    "AFC_AlarmAckn"(trigger := NOT #i.status.vctrl AND #i.out.run,
	                    release := NOT #i.sim.ctrl,
	                    ctrlpoint := FALSE,
	                    enackn := TRUE,
	                    ensiren := TRUE,
	                    p100ms := #p100ms,
	                    generalackn := #generalackn OR #i.faults.fpreset,
	                    reset := #reset OR #i.faults.fpreset,
	                    mute := #mute,
	                    delay := 0.0,
	                    plcackn => #faults.ctrl.plcackn_ctrl,
	                    alarm => #faults.ctrl.alarm_ctrl,
	                    siren => #faults.status.siren_ctrl,
	                    hmiackn := #faults.status.hmiackn_ctrl,
	                    Data := #i.faults.ctrl);
	    
	    //Network8: FAULT: Interlock violation
	    
	    "AFC_AlarmAckn"(trigger := #start AND #block,
	                    release := #i.status.ilstart,
	                    ctrlpoint := FALSE,
	                    enackn := TRUE,
	                    ensiren := TRUE,
	                    p100ms := #p100ms,
	                    generalackn := #generalackn OR #i.faults.fpreset,
	                    reset := #reset OR #i.faults.fpreset,
	                    mute := #mute,
	                    delay := 0.0,
	                    plcackn => #faults.ctrl.plcackn_il,
	                    alarm => #faults.ctrl.alarm_il,
	                    siren => #faults.status.siren_il,
	                    hmiackn := #faults.status.hmiackn_il,
	                    Data := #i.faults.il);
	    
	END_REGION
	
	REGION STATUS  NW:9-10
	    
	    //Network9: STATUS: General Fault
	    
	    #i.status.fault := #i.faults.ftr.status.alarm OR #i.faults.fts.status.alarm OR #i.faults.mcb.status.alarm OR #i.faults.ctrl.status.alarm OR #i.faults.il.status.alarm;
	    
	    //Network10: STATUS: Start interlock
	    
	    #i.status.ilstart := NOT (#block OR #i.status.fault) AND #i.status.vctrl;
	    
	END_REGION
	
	REGION CONTROL  NW:11-13
	    
	    //Network11: CONTROL: Manual Set
	    
	    #condSET := #i.cmd.man OR #manualset;
	    #condRESET := #i.cmd.auto OR #autoset;
	    
	    #i.ind.man := (#i.ind.man OR #condSET) AND NOT #condRESET;
	    
	    //Network12: CONTROL: Auto Set
	    
	    #i.ind.auto := NOT #i.ind.man;
	    
	    //Network13: CONTROL: Manual Run
	    
	    #condSET := #i.cmd.start AND #i.ind.man;
	    #condRESET := #i.cmd.stop OR NOT (#i.ind.man AND #i.status.ilstart);
	    
	    #i.out.manrun := (#i.out.manrun OR #condSET) AND NOT #condRESET;
	    
	END_REGION
	
	REGION STATUS  NW:14-15
	    
	    //Network14: STATUS: Motor's icon
	    
	    #i.status.icon := 0;
	    
	    IF #i.status.vfb AND NOT #i.status.fault AND #i.status.vctrl
	    THEN
	        #i.status.icon := 1;
	    ELSIF #i.status.vfb AND NOT #i.status.fault AND NOT #i.status.vctrl
	    THEN
	        #i.status.icon := 2;
	    ELSIF #i.status.fault AND #blink
	    THEN
	        #i.status.icon := 3;
	    END_IF;
	    
	    //Network15: STATUS:Start/Stop Buttons
	    
	    #i.ind.start := #i.out.manrun AND #i.ind.man;
	    #i.ind.stop := NOT #i.out.manrun AND #i.ind.man;
	    
	END_REGION
	
	REGION OUTPUT  NW:16
	    
	    //Network16: OUTPUT: Start motor
	    
	     #condSET := #i.status.ilstart AND (#i.out.manrun OR (#start AND #i.ind.auto));
	    #condRESET := NOT #i.status.ilstart;
	    
	    "AFC_DelayONOFF"(cmd := #condSET,
	                     Pulse := #p100ms,
	                     Reset := #condRESET,
	                     on => #i.out.run,
	                     Data := #i.delay);
	    
	END_REGION
	
	REGION MNT  NW:17-19
	    
	    //Network17: ARH: Working hours counter
	    
	    IF #i.status.vfb AND #p1s THEN
	        #i.arh.seconds := #i.arh.seconds + 1;
	    END_IF;
	    
	    #i.arh.hour := #i.arh.seconds >= 3600;
	    
	    IF #i.arh.hour THEN
	        #i.arh.actual := #i.arh.actual + 1;
	        #i.arh.seconds := 0;
	    END_IF;
	    
	    IF #i.arh.resetarh THEN
	        #i.arh.actual := #i.arh.lastmaint := 0;
	    END_IF;
	    
	    #i.arh.difference := #i.arh.actual - #i.arh.lastmaint;
	    
	    //Network18: ARH: Maintenance required
	    
	    #condSET := #i.arh.difference >= #i.arh.checkafter;
	    #condRESET := (#i.arh.completed AND #i.arh.maintenance) OR NOT #i.arh.enable;
	    
	    #i.arh.maintenance := (#i.arh.maintenance OR #condSET) AND NOT #condRESET;
	    
	    IF #i.arh.completed AND #i.arh.maintenance THEN
	        #i.arh.lastmaint := #i.arh.actual;
	    END_IF;
	    
	    //Network19: STATUS: Maintenance required
	    
	    #i.status.maint := #i.arh.maintenance;
	    
	END_REGION
	
	REGION OUTPUT  NW:20
	    
	    //Network20: Move UDT outputs to FC outputs
	    
	    #run := #i.out.run;
	    #vfb := #i.status.vfb;
	    
	END_REGION
	
	REGION BUTTON  NW:21
	    
	    //Network21: EXTRA: Button treatment
	    
	    IF #i.ind.auto THEN
	        #i.cmd.auto := FALSE;
	    END_IF;
	    
	    IF #i.ind.man THEN
	        #i.cmd.man := FALSE;
	    END_IF;
	    
	    IF #i.ind.start OR #i.ind.auto OR NOT #i.status.ilstart THEN
	        #i.cmd.start := FALSE;
	    END_IF;
	    
	    IF #i.ind.stop OR #i.ind.auto THEN
	        #i.cmd.stop := FALSE;
	    END_IF;
	    
	    IF #i.faults.fpreset THEN
	        #i.faults.fpreset := FALSE;
	    END_IF;
	    
	    IF (#i.arh.seconds = 0) AND (#i.arh.actual = 0) THEN
	        #i.arh.resetarh := FALSE;
	    END_IF;
	    
	END_REGION
END_FUNCTION_BLOCK

FUNCTION_BLOCK "AFB_MotorLinearCtrl_v3"
{ S7_Optimized_Access := 'TRUE' }
VERSION : 0.1
   VAR_INPUT 
      start { ExternalAccessible := 'False'; ExternalVisible := 'False'; ExternalWritable := 'False'} : Bool;   // "Logic" in order to start
      followup { ExternalAccessible := 'False'; ExternalVisible := 'False'; ExternalWritable := 'False'} : Bool;   // 0=motor control from PID, 1=motor setpoint directly from program
      "fb" { ExternalAccessible := 'False'; ExternalVisible := 'False'; ExternalWritable := 'False'} : Bool;   // Motor's running feedback (1=run, 0=stop)
      mcb { ExternalAccessible := 'False'; ExternalVisible := 'False'; ExternalWritable := 'False'} : Bool;   // Motor circuit breaker (1=ok, 0=fault)
      ctrl { ExternalAccessible := 'False'; ExternalVisible := 'False'; ExternalWritable := 'False'} : Bool;   // Control of motor (1=PLC, 0=Local)
      vfdnotrip { ExternalAccessible := 'False'; ExternalVisible := 'False'; ExternalWritable := 'False'} : Bool;   // VFD health condition (1=ok, 0=fault)
      block { ExternalAccessible := 'False'; ExternalVisible := 'False'; ExternalWritable := 'False'} : Bool;   // Condition that blocks motor operation
      generalackn { ExternalAccessible := 'False'; ExternalVisible := 'False'; ExternalWritable := 'False'} : Bool;   // General acknowledgement
      reset { ExternalAccessible := 'False'; ExternalVisible := 'False'; ExternalWritable := 'False'} : Bool;   // Option that resets the faults
      mute { ExternalAccessible := 'False'; ExternalVisible := 'False'; ExternalWritable := 'False'} : Bool;   // Mute siren
      autoset { ExternalAccessible := 'False'; ExternalVisible := 'False'; ExternalWritable := 'False'} : Bool;   // Option that sets the motor to auto mode (Used for mass auto set)
      manualset { ExternalAccessible := 'False'; ExternalVisible := 'False'; ExternalWritable := 'False'} : Bool;   // Option that sets the motor to manual mode (Used for mass manual set)
      p1s { ExternalAccessible := 'False'; ExternalVisible := 'False'; ExternalWritable := 'False'} : Bool;   // Pulse that is generated every 1 s (Count up)
      p100ms { ExternalAccessible := 'False'; ExternalVisible := 'False'; ExternalWritable := 'False'} : Bool;   // Pulse that is generated every 100 ms (Count up)
      blink { ExternalAccessible := 'False'; ExternalVisible := 'False'; ExternalWritable := 'False'} : Bool;   // Blink that is used for the graphics (Frequency of CPU)
      PV { ExternalAccessible := 'False'; ExternalVisible := 'False'; ExternalWritable := 'False'} : Real;   // Peripheral value as independent variable to the linear controller
      PV_unit { ExternalAccessible := 'False'; ExternalVisible := 'False'; ExternalWritable := 'False'} : WString;   // Peripheral value unit
      FUP { ExternalAccessible := 'False'; ExternalVisible := 'False'; ExternalWritable := 'False'} : Real;   // Follow up value
      Out_unit { ExternalAccessible := 'False'; ExternalVisible := 'False'; ExternalWritable := 'False'} : WString;   // Output unit (If nothing is entered then it is from the HMI)
   END_VAR

   VAR_OUTPUT 
      run { ExternalAccessible := 'False'; ExternalVisible := 'False'; ExternalWritable := 'False'} : Bool;   // Command to start motor
      vfb { ExternalAccessible := 'False'; ExternalVisible := 'False'; ExternalWritable := 'False'} : Bool;   // Virtual feedback (used everywhere instead of digital fb)
      reference { ExternalAccessible := 'False'; ExternalVisible := 'False'; ExternalWritable := 'False'} : Int;   // Reference to analog output card
   END_VAR

   VAR_IN_OUT 
      faults : "UDT_MTRFAULTS";   // External data (Primary alarm data - alarm & plc ackn)
   END_VAR

   VAR RETAIN
      i : "UDT_MOTORLINEAR";   // Data type containing the motor's data
   END_VAR
   VAR 
      calc { ExternalAccessible := 'False'; ExternalVisible := 'False'; ExternalWritable := 'False'} : Struct   // Calculations for scaling process
         inspan { ExternalAccessible := 'False'; ExternalVisible := 'False'; ExternalWritable := 'False'} : Real;   // Scaling span
         outspan { ExternalAccessible := 'False'; ExternalVisible := 'False'; ExternalWritable := 'False'} : Real;   // Channel span
         xmax { ExternalAccessible := 'False'; ExternalVisible := 'False'; ExternalWritable := 'False'} : Real;   // Channel maximum value
         xmin { ExternalAccessible := 'False'; ExternalVisible := 'False'; ExternalWritable := 'False'} : Real;   // Channel minimum value
         ymax { ExternalAccessible := 'False'; ExternalVisible := 'False'; ExternalWritable := 'False'} : Real;   // Output maximum value
         ymin { ExternalAccessible := 'False'; ExternalVisible := 'False'; ExternalWritable := 'False'} : Real;   // Output minimum value
         x { ExternalAccessible := 'False'; ExternalVisible := 'False'; ExternalWritable := 'False'} : Real;   // Active x value (channel)
         y { ExternalAccessible := 'False'; ExternalVisible := 'False'; ExternalWritable := 'False'} : Real;   // Active y value (output)
         speedmin { ExternalAccessible := 'False'; ExternalVisible := 'False'; ExternalWritable := 'False'} : Real;   // Minimum speed
         speedmax { ExternalAccessible := 'False'; ExternalVisible := 'False'; ExternalWritable := 'False'} : Real;   // Maximum speed
         sign { ExternalAccessible := 'False'; ExternalVisible := 'False'; ExternalWritable := 'False'} : Bool;   // Linear scaling slope sign
      END_STRUCT;
   END_VAR

   VAR_TEMP 
      ctrl_internal : Bool;   // Internal control (0=follow up, 1=linear)
      condSET : Bool;
      condRESET : Bool;
   END_VAR


BEGIN
	REGION GEN  NW:2
	    
	    //Network2: GEN: Move FB inputs to UDT inputs
	    
	    #ctrl_internal := NOT #followup AND #i.ctrl.linear;
	    #i.ctrl.PV := #PV;
	    #i.ctrl.FUP := #FUP;
	    #i.ctrl.pvunit := #PV_unit;
	    
	    IF #Out_unit <> WSTRING#'' THEN
	        #i.ctrl.outunit := #Out_unit;
	    END_IF;
	    
	END_REGION
	
	REGION STATUS  NW:3-4
	    
	    //Network3: STATUS: Virtual feedback
	    
	    #i.status.vfb := (#fb AND NOT #i.sim.fb) OR (#i.out.run AND #i.sim.fb);
	    
	    //Network4: STATUS: Virtual control
	    
	    #i.status.vctrl := #i.sim.ctrl OR (#ctrl AND NOT #i.sim.ctrl);
	    
	END_REGION
	
	REGION FAULT  NW:5-10
	    
	    //Network5: FAULT: Fail to run
	    
	    "AFC_AlarmAckn"(trigger := NOT #i.status.vfb AND #i.out.run AND #i.status.vctrl,
	                    release := NOT #i.sim.fb,
	                    ctrlpoint := FALSE,
	                    enackn := TRUE,
	                    ensiren := TRUE,
	                    p100ms := #p100ms,
	                    generalackn := #generalackn OR #i.faults.fpreset,
	                    reset := #reset OR #i.faults.fpreset,
	                    mute := #mute,
	                    delay := 0.0,
	                    plcackn => #faults.ctrl.plcackn_ftr,
	                    alarm => #faults.ctrl.alarm_ftr,
	                    siren => #faults.status.siren_ftr,
	                    hmiackn := #faults.status.hmiackn_ftr,
	                    Data := #i.faults.ftr);
	    
	    //Network6: FAULT: Fail to stop
	    
	    "AFC_AlarmAckn"(trigger := #i.status.vfb AND NOT #i.out.run AND #i.status.vctrl,
	                    release := NOT #i.sim.fb,
	                    ctrlpoint := FALSE,
	                    enackn := TRUE,
	                    ensiren := TRUE,
	                    p100ms := #p100ms,
	                    generalackn := #generalackn OR #i.faults.fpreset,
	                    reset := #reset OR #i.faults.fpreset,
	                    mute := #mute,
	                    delay := 0.0,
	                    plcackn => #faults.ctrl.plcackn_fts,
	                    alarm => #faults.ctrl.alarm_fts,
	                    siren => #faults.status.siren_fts,
	                    hmiackn := #faults.status.hmiackn_fts,
	                    Data := #i.faults.fts);
	    
	    //Network7: FAULT: Monor circuit breaker
	    
	    "AFC_AlarmAckn"(trigger := NOT #mcb,
	                    release := NOT #i.sim.fb,
	                    ctrlpoint := FALSE,
	                    enackn := TRUE,
	                    ensiren := TRUE,
	                    p100ms := #p100ms,
	                    generalackn := #generalackn OR #i.faults.fpreset,
	                    reset := #reset OR #i.faults.fpreset,
	                    mute := #mute,
	                    delay := 0.0,
	                    plcackn => #faults.ctrl.plcackn_mcb,
	                    alarm => #faults.ctrl.alarm_mcb,
	                    siren => #faults.status.siren_mcb,
	                    hmiackn := #faults.status.hmiackn_mcb,
	                    Data := #i.faults.mcb);
	    
	    //Network8: FAULT: Control
	    
	    "AFC_AlarmAckn"(trigger := NOT #i.status.vctrl AND #i.out.run,
	                    release := NOT #i.sim.ctrl,
	                    ctrlpoint := FALSE,
	                    enackn := TRUE,
	                    ensiren := TRUE,
	                    p100ms := #p100ms,
	                    generalackn := #generalackn OR #i.faults.fpreset,
	                    reset := #reset OR #i.faults.fpreset,
	                    mute := #mute,
	                    delay := 0.0,
	                    plcackn => #faults.ctrl.plcackn_ctrl,
	                    alarm => #faults.ctrl.alarm_ctrl,
	                    siren => #faults.status.siren_ctrl,
	                    hmiackn := #faults.status.hmiackn_ctrl,
	                    Data := #i.faults.ctrl);
	    
	    //Network9: FAULT: Variable frequency drive
	    
	    "AFC_AlarmAckn"(trigger := NOT #vfdnotrip,
	                    release := TRUE,
	                    ctrlpoint := FALSE,
	                    enackn := TRUE,
	                    ensiren := TRUE,
	                    p100ms := #p100ms,
	                    generalackn := #generalackn OR #i.faults.fpreset,
	                    reset := #reset OR #i.faults.fpreset,
	                    mute := #mute,
	                    delay := 0.0,
	                    plcackn => #faults.ctrl.plcackn_vfd,
	                    alarm => #faults.ctrl.alarm_vfd,
	                    siren => #faults.status.siren_vfd,
	                    hmiackn := #faults.status.hmiackn_vfd,
	                    Data := #i.faults.vfd);
	    
	    //Network10: FAULT: Interlock violation
	    
	    "AFC_AlarmAckn"(trigger := #start AND #block,
	                    release := #i.status.ilstart,
	                    ctrlpoint := FALSE,
	                    enackn := TRUE,
	                    ensiren := TRUE,
	                    p100ms := #p100ms,
	                    generalackn := #generalackn OR #i.faults.fpreset,
	                    reset := #reset OR #i.faults.fpreset,
	                    mute := #mute,
	                    delay := 0.0,
	                    plcackn => #faults.ctrl.plcackn_il,
	                    alarm => #faults.ctrl.alarm_il,
	                    siren => #faults.status.siren_il,
	                    hmiackn := #faults.status.hmiackn_il,
	                    Data := #i.faults.il);
	    
	END_REGION
	
	REGION STATUS  NW:11-12
	    
	    //Network11: STATUS: General Fault
	    
	    #i.status.fault := #i.faults.ftr.status.alarm OR #i.faults.fts.status.alarm OR #i.faults.mcb.status.alarm OR #i.faults.ctrl.status.alarm OR #i.faults.vfd.status.alarm OR #i.faults.il.status.alarm;
	    
	    //Network12: STATUS: Start interlock
	    
	    #i.status.ilstart := NOT (#block OR #i.status.fault) AND #i.status.vctrl AND #i.unscale.set AND (NOT #ctrl_internal OR #i.scale.set OR #i.ctrl.mode);
	    
	END_REGION
	
	REGION CONTROL  NW:13-15
	    
	    //Network13: CONTROL: Manual Set
	    
	    #condSET := #i.cmd.man OR #manualset;
	    #condRESET := #i.cmd.auto OR #autoset;
	    
	    #i.ind.man := (#i.ind.man OR #condSET) AND NOT #condRESET;
	    
	    //Network14: CONTROL: Auto Set
	    
	    #i.ind.auto := NOT #i.ind.man;
	    
	    //Network15: CONTROL: Manual Run
	    
	    #condSET := #i.cmd.start AND #i.ind.man;
	    #condRESET := #i.cmd.stop OR NOT (#i.ind.man AND #i.status.ilstart);
	    
	    #i.out.manrun := (#i.out.manrun OR #condSET) AND NOT #condRESET;
	    
	END_REGION
	
	REGION STATUS  NW:16-17
	    
	    //Network16: STATUS: Motor's icon
	    
	    #i.status.icon := 0;
	    
	    IF #i.status.vfb AND NOT #i.status.fault AND #i.status.vctrl
	    THEN
	        #i.status.icon := 1;
	    ELSIF #i.status.vfb AND NOT #i.status.fault AND NOT #i.status.vctrl
	    THEN
	        #i.status.icon := 2;
	    ELSIF #i.status.fault AND #blink
	    THEN
	        #i.status.icon := 3;
	    END_IF;
	    
	    //Network17: STATUS:Start/Stop Buttons
	    
	    #i.ind.start := #i.out.manrun AND #i.ind.man;
	    #i.ind.stop := NOT #i.out.manrun AND #i.ind.man;
	    
	END_REGION
	
	REGION OUTPUT  NW:18
	    
	    //Network18: OUTPUT: Start motor
	    
	    #condSET := #i.status.ilstart AND (#i.out.manrun OR (#start AND #i.ind.auto));
	    #condRESET := NOT #i.status.ilstart;
	    
	    "AFC_DelayONOFF"(cmd := #condSET,
	                     Pulse := #p100ms,
	                     Reset := #condRESET,
	                     on => #i.out.run,
	                     Data := #i.delay);
	    
	END_REGION
	
	REGION SCALE  NW:19-22
	    
	    //Network19: SCALE: Move input
	    
	    #i.scale.in := #i.ctrl.PV;
	    
	    //Network20: SCALE: Cross-check unscaling setup
	    
	    #i.scale.set := (#i.scale.instart <> #i.scale.inend) AND (#i.scale.outstart <> #i.scale.outend);
	    
	    //Network21: SCALE: Determine sign of scaling slope and calculation operands (Hi - Low)
	    
	    IF #i.scale.set THEN
	        #calc.inspan := #i.scale.inend - #i.scale.instart;
	        #calc.outspan := #i.scale.outend - #i.scale.outstart;
	        #calc.x := #i.scale.in;
	        IF #calc.inspan > 0 AND #calc.outspan > 0 THEN
	            #calc.sign := TRUE;
	            #calc.ymax := #i.scale.outend;
	            #calc.ymin := #i.scale.outstart;
	            #calc.xmax := #i.scale.inend;
	            #calc.xmin := #i.scale.instart;
	        ELSIF #calc.inspan < 0 AND #calc.outspan < 0 THEN
	            #calc.sign := TRUE;
	            #calc.ymax := #i.scale.outstart;
	            #calc.ymin := #i.scale.outend;
	            #calc.xmax := #i.scale.instart;
	            #calc.xmin := #i.scale.inend;
	        ELSIF #calc.inspan < 0 AND #calc.outspan > 0 THEN
	            #calc.sign := FALSE;
	            #calc.ymax := #i.scale.outstart;
	            #calc.ymin := #i.scale.outend;
	            #calc.xmax := #i.scale.inend;
	            #calc.xmin := #i.scale.instart;
	        ELSE
	            #calc.sign := FALSE;
	            #calc.ymax := #i.scale.outend;
	            #calc.ymin := #i.scale.outstart;
	            #calc.xmax := #i.scale.instart;
	            #calc.xmin := #i.scale.inend;
	        END_IF;
	    ELSE
	        #calc.inspan := #calc.outspan := #calc.xmax := #calc.xmin := #calc.ymax := #calc.ymin := 0;
	    END_IF;
	    
	    //Network22: SCALE: Determine output
	    
	    IF #i.scale.set AND #calc.sign THEN
	        
	        #calc.y := #calc.ymin + ((#calc.ymax - #calc.ymin) * (#calc.x - #calc.xmin) / (#calc.xmax - #calc.xmin));
	        
	        IF #calc.x <= #calc.xmin THEN
	            #calc.y := #calc.ymin;
	        END_IF;
	        
	        IF #calc.x >= #calc.xmax THEN
	            #calc.y := #calc.ymax;
	        END_IF;
	        
	    END_IF;
	    
	    IF #i.scale.set AND NOT #calc.sign THEN
	        
	        #calc.y := #calc.ymin + ((#calc.ymax - #calc.ymin) * (#calc.xmax - #calc.x) / (#calc.xmax - #calc.xmin));
	        
	        IF #calc.x <= #calc.xmin THEN
	            #calc.y := #calc.ymax;
	        END_IF;
	        
	        IF #calc.x >= #calc.xmax THEN
	            #calc.y := #calc.ymin;
	        END_IF;
	        
	    END_IF;
	    
	    IF #i.scale.set THEN
	        #i.scale.output := #calc.y;
	    END_IF;
	    
	END_REGION
	
	REGION SPEED CONTROL  NW:23-27
	    
	    //Network23: SPEED CONTROL: Manage speed control limits
	    
	    IF (#i.ctrl.ITLVAL < #calc.speedmin) AND (#i.ctrl.ITLVAL > #calc.speedmax) THEN
	        #i.ctrl.ITLVAL := #calc.speedmin;
	    END_IF;
	    
